KUKA KRL program: EPS_2_25990_SANMH03_A_20251014010956.src

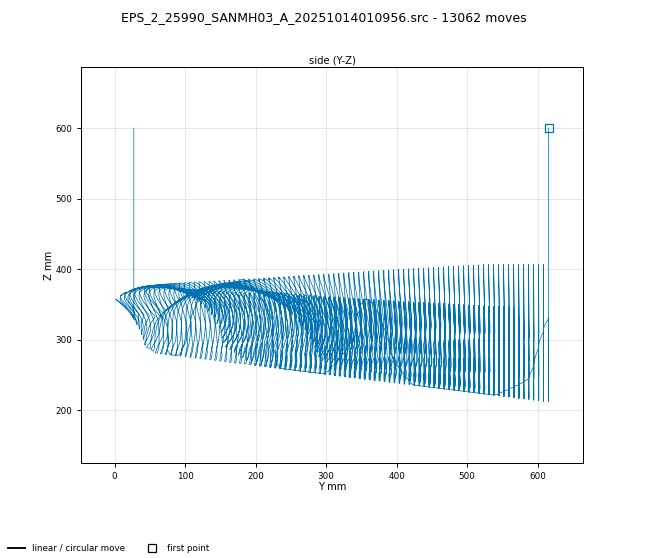
[picture p0: tool path of EPS_2_25990_SANMH03_A_20251014010956.src, 13062 of 13064 moves have a stored position in this frame; points joined in program order, loops and branches not executed]
&ACCESS RVP
&REL 4
&COMMENT QRS 19112012
&PARAM EDITMASK = *
DEF PART()
EXT BAS (BAS_COMMAND :IN,REAL :IN )
INT I
BAS (#INITMOV,0 )

;KUKA QRS Post kuka4.cps  Date:22-06-2017 !

File_ID=2884

QRS_PRE_INIT()

;Init var - Until changes are made in qrs_pre_init
Outlet_Square_prg=0
Inlet_1_Square_prg=0
Inlet_2_Square_prg=0
Inlet_3_Square_prg=0
Inlet_4_Square_prg=0
Inlet_5_Square_prg=0

Outlet_1={X 0.000, Y 531.880, Z 306.500, B 0.000, E1 0.000 }
Inlet_1={X 0.000, Y 536.220, Z 246.500, B 0.000, E1 91.000 }
Inlet_2={X 0.000, Y 540.650, Z 272.000, B 0.000, E1 217.000 }
Outlet_1_type=201
Inlet_1_type=201
Inlet_2_type=150
;QRS#1=Sidecore dimensions
;QRS#2=200-8" PVC SDR 35
;QRS#3=200-8" PVC SDR 35
;QRS#4=150-6" PVC SDR 28
;QRS#5=
;QRS#6=
;QRS#7=
;QRS#8=
;QRS#9=12-08 PSX
;QRS#10=12-08 PSX
;QRS#11=10-06 PSX
;QRS#12=
;QRS#13=
;QRS#14=
;QRS#15=
;QRS#16=1220x127x686 2,25'
;QRS#17=EPS Height
;QRS#18=407
;QRS#19=*
;QRS#20= UPDATED VERSION 22-06-2017
;QRS#21=*
Outlet_Square=0100
Inlet_1_Square=0100
Inlet_2_Square=070
Inlet_3_Square=0
Inlet_4_Square=0
Inlet_5_Square=0
Mill_Square=1
Outlet_Square_Prg=204
Inlet_1_Square_prg=204
Inlet_2_Square_prg=203

QRS_INIT()

$ADVANCE=5

; T1
PTP {E1 173.516,E2 173.516}
PTP {X 0,Y 615.499,A -85,B 0,C 180,E1 173.516,E2 173.516,E3 0,E4 0,E5 0,E6 0}
QRS_SPEED_INIT()
LIN {X 0,Y 615.499,Z 600,A -85,B 0,C 180,E1 173.516,E2 173.516,E3 0,E4 0,E5 0,E6 0} C_VEL
LIN {X 0,Y 615.499,Z 343.49,A -85,B 0,C 180,E1 173.516,E2 173.516} C_VEL
LIN {X 0,Y 615.499,Z 333.343,A -85,B 0,C 180,E1 173.516,E2 173.516} C_VEL
LIN {X 0,Y 615.495,Z 331.594,A -85,B 0,C 180,E1 173.42,E2 173.42} C_VEL
LIN {X 0,Y 615.496,Z 325.468,A -85,B 0,C 180,E1 172.454,E2 172.454} C_VEL
LIN {X 0,Y 615.497,Z 317.616,A -85,B 0,C 180,E1 171.463,E2 171.463} C_VEL
LIN {X 0,Y 615.498,Z 307.826,A -85,B 0,C 180,E1 170.47,E2 170.47} C_VEL
LIN {X 0,Y 615.498,Z 297.546,A -85,B 0,C 180,E1 169.639,E2 169.639} C_VEL
LIN {X 0,Y 615.47,Z 285.87,A -85,B 0,C 180,E1 168.885,E2 168.885} C_VEL
LIN {X 0,Y 615.494,Z 274.386,A -85,B 0,C 180,E1 168.306,E2 168.306} C_VEL
LIN {X 0,Y 615.485,Z 262.385,A -85,B 0,C 180,E1 167.846,E2 167.846} C_VEL
LIN {X 0,Y 615.487,Z 250.236,A -85,B 0,C 180,E1 167.512,E2 167.512} C_VEL
LIN {X 0,Y 615.486,Z 243.189,A -85,B 0,C 180,E1 167.365,E2 167.365} C_VEL
LIN {X 0,Y 615.467,Z 239.503,A -85,B 0,C 180,E1 164.773,E2 164.773} C_VEL
LIN {X 0,Y 615.492,Z 235.664,A -85,B 0,C 180,E1 162.043,E2 162.043} C_VEL
LIN {X 0,Y 615.451,Z 231.833,A -85,B 0,C 180,E1 159.268,E2 159.268} C_VEL
LIN {X 0,Y 615.489,Z 227.979,A -85,B 0,C 180,E1 156.444,E2 156.444} C_VEL
LIN {X 0,Y 615.499,Z 225.095,A -85,B 0,C 180,E1 154.285,E2 154.285} C_VEL
LIN {X 0,Y 615.431,Z 221.535,A -85,B 0,C 180,E1 151.56,E2 151.56} C_VEL
LIN {X 0,Y 615.482,Z 218.202,A -85,B 0,C 180,E1 148.916,E2 148.916} C_VEL
LIN {X 0,Y 615.46,Z 214.61,A -85,B 0,C 180,E1 145.976,E2 145.976} C_VEL
LIN {X 0,Y 615.49,Z 211.697,A -85,B 0,C 180,E1 143.575,E2 143.575} C_VEL
LIN {X 0,Y 615.494,Z 211.683,A -85,B 0,C 180,E1 140.938,E2 140.938} C_VEL
LIN {X 0,Y 615.476,Z 211.697,A -85,B 0,C 180,E1 137.922,E2 137.922} C_VEL
LIN {X 0,Y 615.492,Z 211.687,A -85,B 0,C 180,E1 135.069,E2 135.069} C_VEL
LIN {X 0,Y 615.464,Z 211.698,A -85,B 0,C 180,E1 132.355,E2 132.355} C_VEL
LIN {X 0,Y 615.436,Z 211.697,A -85,B 0,C 180,E1 129.755,E2 129.755} C_VEL
LIN {X 0,Y 615.487,Z 211.699,A -85,B 0,C 180,E1 127.243,E2 127.243} C_VEL
LIN {X 0,Y 615.44,Z 211.698,A -85,B 0,C 180,E1 124.694,E2 124.694} C_VEL
LIN {X 0,Y 615.438,Z 211.697,A -85,B 0,C 180,E1 122.323,E2 122.323} C_VEL
LIN {X 0,Y 615.495,Z 211.7,A -85,B 0,C 180,E1 119.795,E2 119.795} C_VEL
LIN {X 0,Y 615.469,Z 211.689,A -85,B 0,C 180,E1 117.041,E2 117.041} C_VEL
LIN {X 0,Y 615.487,Z 211.702,A -85,B 0,C 180,E1 114.272,E2 114.272} C_VEL
LIN {X 0,Y 615.493,Z 211.684,A -85,B 0,C 180,E1 111.432,E2 111.432} C_VEL
LIN {X 0,Y 615.485,Z 211.699,A -85,B 0,C 180,E1 108.603,E2 108.603} C_VEL
LIN {X 0,Y 615.477,Z 211.687,A -85,B 0,C 180,E1 105.906,E2 105.906} C_VEL
LIN {X 0,Y 615.495,Z 211.701,A -85,B 0,C 180,E1 103.201,E2 103.201} C_VEL
LIN {X 0,Y 615.441,Z 211.696,A -85,B 0,C 180,E1 100.528,E2 100.528} C_VEL
LIN {X 0,Y 615.484,Z 211.697,A -85,B 0,C 180,E1 97.876,E2 97.876} C_VEL
LIN {X 0,Y 615.432,Z 211.7,A -85,B 0,C 180,E1 95.242,E2 95.242} C_VEL
LIN {X 0,Y 615.433,Z 211.698,A -85,B 0,C 180,E1 93.273,E2 93.273} C_VEL
LIN {X 0,Y 615.439,Z 211.696,A -85,B 0,C 180,E1 91.309,E2 91.309} C_VEL
LIN {X 0,Y 615.472,Z 211.699,A -85,B 0,C 180,E1 88.691,E2 88.691} C_VEL
LIN {X 0,Y 615.487,Z 211.688,A -85,B 0,C 180,E1 86.072,E2 86.072} C_VEL
LIN {X 0,Y 615.477,Z 211.777,A -85,B 0,C 180,E1 85.005,E2 85.005} C_VEL
LIN {X 0,Y 615.488,Z 217.2,A -85,B 0,C 180,E1 82.784,E2 82.784} C_VEL
LIN {X 0,Y 615.49,Z 223.43,A -85,B 0,C 180,E1 80.138,E2 80.138} C_VEL
LIN {X 0,Y 615.452,Z 229.574,A -85,B 0,C 180,E1 77.469,E2 77.469} C_VEL
LIN {X 0,Y 615.493,Z 235.878,A -85,B 0,C 180,E1 74.774,E2 74.774} C_VEL
LIN {X 0,Y 615.474,Z 242.411,A -85,B 0,C 180,E1 72.043,E2 72.043} C_VEL
LIN {X 0,Y 615.487,Z 249.137,A -85,B 0,C 180,E1 69.269,E2 69.269} C_VEL
LIN {X 0,Y 615.485,Z 256.099,A -85,B 0,C 180,E1 66.444,E2 66.444} C_VEL
LIN {X 0,Y 615.479,Z 263.285,A -85,B 0,C 180,E1 63.555,E2 63.555} C_VEL
LIN {X 0,Y 615.49,Z 266.918,A -85,B 0,C 180,E1 62.108,E2 62.108} C_VEL
LIN {X 0,Y 615.488,Z 278.231,A -85,B 0,C 180,E1 61.82,E2 61.82} C_VEL
LIN {X 0,Y 615.464,Z 288.228,A -85,B 0,C 180,E1 61.447,E2 61.447} C_VEL
LIN {X 0,Y 615.467,Z 296.234,A -85,B 0,C 180,E1 61.061,E2 61.061} C_VEL
LIN {X 0,Y 615.491,Z 304.039,A -85,B 0,C 180,E1 60.594,E2 60.594} C_VEL
LIN {X 0,Y 615.496,Z 311.816,A -85,B 0,C 180,E1 60.023,E2 60.023} C_VEL
LIN {X 0,Y 615.498,Z 318.16,A -85,B 0,C 180,E1 59.461,E2 59.461} C_VEL
LIN {X 0,Y 615.498,Z 324.688,A -85,B 0,C 180,E1 58.764,E2 58.764} C_VEL
LIN {X 0,Y 615.496,Z 330.585,A -85,B 0,C 180,E1 57.992,E2 57.992} C_VEL
LIN {X 0,Y 615.493,Z 335.716,A -85,B 0,C 180,E1 57.154,E2 57.154} C_VEL
LIN {X 0,Y 615.494,Z 339.016,A -85,B 0,C 180,E1 56.466,E2 56.466} C_VEL
LIN {X 0,Y 615.494,Z 343.165,A -85,B 0,C 180,E1 55.299,E2 55.299} C_VEL
LIN {X 0,Y 615.492,Z 345.468,A -85,B 0,C 180,E1 54.166,E2 54.166} C_VEL
LIN {X 0,Y 615.495,Z 346.361,A -85,B 0,C 180,E1 53.063,E2 53.063} C_VEL
LIN {X 0,Y 615.491,Z 345.737,A -85,B 0,C 180,E1 51.932,E2 51.932} C_VEL
LIN {X 0,Y 615.499,Z 343.952,A -85,B 0,C 180,E1 50.937,E2 50.937} C_VEL
LIN {X 0,Y 615.498,Z 340.875,A -85,B 0,C 180,E1 49.91,E2 49.91} C_VEL
LIN {X 0,Y 615.493,Z 336.533,A -85,B 0,C 180,E1 48.905,E2 48.905} C_VEL
LIN {X 0,Y 615.497,Z 330.597,A -85,B 0,C 180,E1 47.919,E2 47.919} C_VEL
LIN {X 0,Y 615.497,Z 324.524,A -85,B 0,C 180,E1 47.127,E2 47.127} C_VEL
LIN {X 0,Y 615.495,Z 319.388,A -85,B 0,C 180,E1 46.568,E2 46.568} C_VEL
LIN {X 0,Y 615.496,Z 313.223,A -85,B 0,C 180,E1 46.002,E2 46.002} C_VEL
LIN {X 0,Y 615.484,Z 306.158,A -85,B 0,C 180,E1 45.46,E2 45.46} C_VEL
LIN {X 0,Y 615.495,Z 298.933,A -85,B 0,C 180,E1 45.001,E2 45.001} C_VEL
LIN {X 0,Y 615.477,Z 291.057,A -85,B 0,C 180,E1 44.59,E2 44.59} C_VEL
LIN {X 0,Y 615.481,Z 282.81,A -85,B 0,C 180,E1 44.248,E2 44.248} C_VEL
LIN {X 0,Y 615.485,Z 273.161,A -85,B 0,C 180,E1 43.95,E2 43.95} C_VEL
LIN {X 0,Y 615.486,Z 266.876,A -85,B 0,C 180,E1 43.785,E2 43.785} C_VEL
LIN {X 0,Y 615.486,Z 260.138,A -85,B 0,C 180,E1 41.094,E2 41.094} C_VEL
LIN {X 0,Y 615.487,Z 253.669,A -85,B 0,C 180,E1 38.486,E2 38.486} C_VEL
LIN {X 0,Y 615.459,Z 247.171,A -85,B 0,C 180,E1 35.83,E2 35.83} C_VEL
LIN {X 0,Y 615.489,Z 240.885,A -85,B 0,C 180,E1 33.236,E2 33.236} C_VEL
LIN {X 0,Y 615.487,Z 235.37,A -85,B 0,C 180,E1 30.92,E2 30.92} C_VEL
LIN {X 0,Y 615.433,Z 229.578,A -85,B 0,C 180,E1 28.441,E2 28.441} C_VEL
LIN {X 0,Y 615.426,Z 224.987,A -85,B 0,C 180,E1 26.447,E2 26.447} C_VEL
LIN {X 0,Y 615.491,Z 219.28,A -85,B 0,C 180,E1 24.008,E2 24.008} C_VEL
LIN {X 0,Y 615.498,Z 212.782,A -85,B 0,C 180,E1 21.432,E2 21.432} C_VEL
LIN {X 0,Y 615.476,Z 211.7,A -85,B 0,C 180,E1 20.994,E2 20.994} C_VEL
LIN {X 0,Y 615.475,Z 211.7,A -85,B 0,C 180,E1 18.6,E2 18.6} C_VEL
LIN {X 0,Y 615.485,Z 211.696,A -85,B 0,C 180,E1 15.905,E2 15.905} C_VEL
LIN {X 0,Y 615.485,Z 211.699,A -85,B 0,C 180,E1 13.201,E2 13.201} C_VEL
LIN {X 0,Y 615.489,Z 211.701,A -85,B 0,C 180,E1 10.527,E2 10.527} C_VEL
LIN {X 0,Y 615.493,Z 211.696,A -85,B 0,C 180,E1 7.876,E2 7.876} C_VEL
LIN {X 0,Y 615.467,Z 211.7,A -85,B 0,C 180,E1 5.241,E2 5.241} C_VEL
LIN {X 0,Y 615.471,Z 211.7,A -85,B 0,C 180,E1 2.618,E2 2.618} C_VEL
LIN {X 0,Y 615.49,Z 211.7,A -85,B 0,C 180,E1 0,E2 0} C_VEL
LIN {X 0,Y 615.488,Z 211.7,A -85,B 0,C 180,E1 -2.618,E2 -2.618} C_VEL
LIN {X 0,Y 615.478,Z 211.699,A -85,B 0,C 180,E1 -5.241,E2 -5.241} C_VEL
LIN {X 0,Y 615.492,Z 211.695,A -85,B 0,C 180,E1 -7.876,E2 -7.876} C_VEL
LIN {X 0,Y 615.489,Z 211.701,A -85,B 0,C 180,E1 -10.887,E2 -10.887} C_VEL
LIN {X 0,Y 615.49,Z 211.695,A -85,B 0,C 180,E1 -13.932,E2 -13.932} C_VEL
LIN {X 0,Y 615.485,Z 211.7,A -85,B 0,C 180,E1 -16.587,E2 -16.587} C_VEL
LIN {X 0,Y 615.496,Z 211.697,A -85,B 0,C 180,E1 -19.338,E2 -19.338} C_VEL
LIN {X 0,Y 615.472,Z 211.7,A -85,B 0,C 180,E1 -22.342,E2 -22.342} C_VEL
LIN {X 0,Y 615.491,Z 211.7,A -85,B 0,C 180,E1 -24.992,E2 -24.992} C_VEL
LIN {X 0,Y 615.48,Z 211.699,A -85,B 0,C 180,E1 -27.178,E2 -27.178} C_VEL
LIN {X 0,Y 615.498,Z 211.699,A -85,B 0,C 180,E1 -29.796,E2 -29.796} C_VEL
LIN {X 0,Y 615.482,Z 211.699,A -85,B 0,C 180,E1 -32.458,E2 -32.458} C_VEL
LIN {X 0,Y 615.491,Z 211.698,A -85,B 0,C 180,E1 -34.815,E2 -34.815} C_VEL
LIN {X 0,Y 615.493,Z 211.696,A -85,B 0,C 180,E1 -37.242,E2 -37.242} C_VEL
LIN {X 0,Y 615.468,Z 211.7,A -85,B 0,C 180,E1 -40.087,E2 -40.087} C_VEL
LIN {X 0,Y 615.465,Z 211.701,A -85,B 0,C 180,E1 -42.355,E2 -42.355} C_VEL
LIN {X 0,Y 615.497,Z 211.696,A -85,B 0,C 180,E1 -45.068,E2 -45.068} C_VEL
LIN {X 0,Y 615.476,Z 211.701,A -85,B 0,C 180,E1 -47.921,E2 -47.921} C_VEL
LIN {X 0,Y 615.498,Z 211.695,A -85,B 0,C 180,E1 -50.937,E2 -50.937} C_VEL
LIN {X 0,Y 615.486,Z 211.702,A -85,B 0,C 180,E1 -53.575,E2 -53.575} C_VEL
LIN {X 0,Y 615.472,Z 211.749,A -85,B 0,C 180,E1 -54.483,E2 -54.483} C_VEL
LIN {X 0,Y 615.478,Z 220.573,A -85,B 0,C 180,E1 -57.153,E2 -57.153} C_VEL
LIN {X 0,Y 615.453,Z 229.832,A -85,B 0,C 180,E1 -59.838,E2 -59.838} C_VEL
LIN {X 0,Y 615.492,Z 239.075,A -85,B 0,C 180,E1 -62.455,E2 -62.455} C_VEL
LIN {X 0,Y 615.456,Z 248.32,A -85,B 0,C 180,E1 -65.007,E2 -65.007} C_VEL
LIN {X 0,Y 615.473,Z 258.107,A -85,B 0,C 180,E1 -67.658,E2 -67.658} C_VEL
LIN {X 0,Y 615.487,Z 268.102,A -85,B 0,C 180,E1 -70.315,E2 -70.315} C_VEL
LIN {X 0,Y 615.486,Z 278.641,A -85,B 0,C 180,E1 -73.072,E2 -73.072} C_VEL
LIN {X 0,Y 615.464,Z 289.077,A -85,B 0,C 180,E1 -75.761,E2 -75.761} C_VEL
LIN {X 0,Y 615.498,Z 299.209,A -85,B 0,C 180,E1 -78.348,E2 -78.348} C_VEL
LIN {X 0,Y 615.497,Z 313.822,A -85,B 0,C 180,E1 -78.64,E2 -78.64} C_VEL
LIN {X 0,Y 615.453,Z 326.972,A -85,B 0,C 180,E1 -79.051,E2 -79.051} C_VEL
LIN {X 0,Y 615.442,Z 338.774,A -85,B 0,C 180,E1 -79.556,E2 -79.556} C_VEL
LIN {X 0,Y 615.489,Z 349.388,A -85,B 0,C 180,E1 -80.138,E2 -80.138} C_VEL
LIN {X 0,Y 615.498,Z 360.232,A -85,B 0,C 180,E1 -80.884,E2 -80.884} C_VEL
LIN {X 0,Y 615.497,Z 370.812,A -85,B 0,C 180,E1 -81.794,E2 -81.794} C_VEL
LIN {X 0,Y 615.498,Z 378.607,A -85,B 0,C 180,E1 -82.62,E2 -82.62} C_VEL
LIN {X 0,Y 615.496,Z 386.203,A -85,B 0,C 180,E1 -83.608,E2 -83.608} C_VEL
LIN {X 0,Y 615.498,Z 393.205,A -85,B 0,C 180,E1 -84.759,E2 -84.759} C_VEL
LIN {X 0,Y 615.494,Z 397.852,A -85,B 0,C 180,E1 -85.744,E2 -85.744} C_VEL
LIN {X 0,Y 615.494,Z 401.399,A -85,B 0,C 180,E1 -86.727,E2 -86.727} C_VEL
LIN {X 0,Y 615.497,Z 403.233,A -85,B 0,C 180,E1 -87.382,E2 -87.382} C_VEL
LIN {X 0,Y 615.5,Z 404.608,A -85,B 0,C 180,E1 -88.037,E2 -88.037} C_VEL
LIN {X 0,Y 615.496,Z 406.174,A -85,B 0,C 180,E1 -89.346,E2 -89.346} C_VEL
LIN {X 0,Y 615.494,Z 406.389,A -85,B 0,C 180,E1 -90,E2 -90} C_VEL
LIN {X 0,Y 615.495,Z 405.58,A -85,B 0,C 180,E1 -91.309,E2 -91.309} C_VEL
LIN {X 0,Y 615.5,Z 404.607,A -85,B 0,C 180,E1 -91.963,E2 -91.963} C_VEL
LIN {X 0,Y 615.497,Z 403.233,A -85,B 0,C 180,E1 -92.618,E2 -92.618} C_VEL
LIN {X 0,Y 615.496,Z 400.349,A -85,B 0,C 180,E1 -93.601,E2 -93.601} C_VEL
LIN {X 0,Y 615.498,Z 396.441,A -85,B 0,C 180,E1 -94.585,E2 -94.585} C_VEL
LIN {X 0,Y 615.499,Z 391.404,A -85,B 0,C 180,E1 -95.57,E2 -95.57} C_VEL
LIN {X 0,Y 615.497,Z 384.869,A -85,B 0,C 180,E1 -96.583,E2 -96.583} C_VEL
LIN {X 0,Y 615.497,Z 377.132,A -85,B 0,C 180,E1 -97.546,E2 -97.546} C_VEL
LIN {X 0,Y 615.498,Z 369.043,A -85,B 0,C 180,E1 -98.371,E2 -98.371} C_VEL
LIN {X 0,Y 615.499,Z 359.165,A -85,B 0,C 180,E1 -99.199,E2 -99.199} C_VEL
LIN {X 0,Y 615.479,Z 347.98,A -85,B 0,C 180,E1 -99.946,E2 -99.946} C_VEL
LIN {X 0,Y 615.441,Z 337.026,A -85,B 0,C 180,E1 -100.528,E2 -100.528} C_VEL
LIN {X 0,Y 615.459,Z 324.774,A -85,B 0,C 180,E1 -101.031,E2 -101.031} C_VEL
LIN {X 0,Y 615.498,Z 312.055,A -85,B 0,C 180,E1 -101.402,E2 -101.402} C_VEL
LIN {X 0,Y 615.498,Z 299.208,A -85,B 0,C 180,E1 -101.652,E2 -101.652} C_VEL
LIN {X 0,Y 615.464,Z 289.077,A -85,B 0,C 180,E1 -104.239,E2 -104.239} C_VEL
LIN {X 0,Y 615.486,Z 278.64,A -85,B 0,C 180,E1 -106.929,E2 -106.929} C_VEL
LIN {X 0,Y 615.487,Z 268.101,A -85,B 0,C 180,E1 -109.685,E2 -109.685} C_VEL
LIN {X 0,Y 615.476,Z 258.104,A -85,B 0,C 180,E1 -112.343,E2 -112.343} C_VEL
LIN {X 0,Y 615.456,Z 248.32,A -85,B 0,C 180,E1 -114.993,E2 -114.993} C_VEL
LIN {X 0,Y 615.448,Z 237.758,A -85,B 0,C 180,E1 -117.917,E2 -117.917} C_VEL
LIN {X 0,Y 615.464,Z 228.484,A -85,B 0,C 180,E1 -120.541,E2 -120.541} C_VEL
LIN {X 0,Y 615.486,Z 220.546,A -85,B 0,C 180,E1 -122.846,E2 -122.846} C_VEL
LIN {X 0,Y 615.492,Z 213.086,A -85,B 0,C 180,E1 -125.215,E2 -125.215} C_VEL
LIN {X 0,Y 615.47,Z 211.7,A -85,B 0,C 180,E1 -125.724,E2 -125.724} C_VEL
LIN {X 0,Y 615.479,Z 211.701,A -85,B 0,C 180,E1 -128.07,E2 -128.07} C_VEL
LIN {X 0,Y 615.488,Z 211.694,A -85,B 0,C 180,E1 -131.094,E2 -131.094} C_VEL
LIN {X 0,Y 615.482,Z 211.7,A -85,B 0,C 180,E1 -133.997,E2 -133.997} C_VEL
LIN {X 0,Y 615.492,Z 211.697,A -85,B 0,C 180,E1 -136.953,E2 -136.953} C_VEL
LIN {X 0,Y 615.48,Z 211.701,A -85,B 0,C 180,E1 -139.393,E2 -139.393} C_VEL
LIN {X 0,Y 615.483,Z 211.699,A -85,B 0,C 180,E1 -141.989,E2 -141.989} C_VEL
LIN {X 0,Y 615.496,Z 211.699,A -85,B 0,C 180,E1 -144.385,E2 -144.385} C_VEL
LIN {X 0,Y 615.487,Z 211.698,A -85,B 0,C 180,E1 -145.3,E2 -145.3} C_VEL
LIN {X 0,Y 615.466,Z 214.459,A -85,B 0,C 180,E1 -147.673,E2 -147.673} C_VEL
LIN {X 0,Y 615.453,Z 217.446,A -85,B 0,C 180,E1 -150.212,E2 -150.212} C_VEL
LIN {X 0,Y 615.448,Z 220.642,A -85,B 0,C 180,E1 -152.963,E2 -152.963} C_VEL
LIN {X 0,Y 615.445,Z 223.297,A -85,B 0,C 180,E1 -155.006,E2 -155.006} C_VEL
LIN {X 0,Y 615.436,Z 226.139,A -85,B 0,C 180,E1 -157.153,E2 -157.153} C_VEL
LIN {X 0,Y 615.435,Z 229.243,A -85,B 0,C 180,E1 -159.457,E2 -159.457} C_VEL
LIN {X 0,Y 615.494,Z 232.768,A -85,B 0,C 180,E1 -162.043,E2 -162.043} C_VEL
LIN {X 0,Y 615.458,Z 236.563,A -85,B 0,C 180,E1 -164.773,E2 -164.773} C_VEL
LIN {X 0,Y 615.474,Z 240.371,A -85,B 0,C 180,E1 -167.47,E2 -167.47} C_VEL
LIN {X 0,Y 615.484,Z 243.185,A -85,B 0,C 180,E1 -169.451,E2 -169.451} C_VEL
LIN {X 0,Y 615.487,Z 258.21,A -85,B 0,C 180,E1 -169.806,E2 -169.806} C_VEL
LIN {X 0,Y 615.491,Z 270.248,A -85,B 0,C 180,E1 -170.221,E2 -170.221} C_VEL
LIN {X 0,Y 615.463,Z 282.68,A -85,B 0,C 180,E1 -170.801,E2 -170.801} C_VEL
LIN {X 0,Y 615.49,Z 293.753,A -85,B 0,C 180,E1 -171.463,E2 -171.463} C_VEL
LIN {X 0,Y 615.498,Z 302.72,A -85,B 0,C 180,E1 -172.125,E2 -172.125} C_VEL
LIN {X 0,Y 615.499,Z 311.875,A -85,B 0,C 180,E1 -172.943,E2 -172.943} C_VEL
LIN {X 0,Y 615.497,Z 320.848,A -85,B 0,C 180,E1 -173.937,E2 -173.937} C_VEL
LIN {X 0,Y 615.497,Z 328.03,A -85,B 0,C 180,E1 -174.923,E2 -174.923} C_VEL
LIN {X 0,Y 615.493,Z 332.875,A -85,B 0,C 180,E1 -175.744,E2 -175.744} C_VEL
LIN {X 0,Y 615.496,Z 337.586,A -85,B 0,C 180,E1 -176.727,E2 -176.727} C_VEL
LIN {X 0,Y 615.498,Z 341.198,A -85,B 0,C 180,E1 -177.71,E2 -177.71} C_VEL
LIN {X 0,Y 615.496,Z 343.818,A -85,B 0,C 180,E1 -178.691,E2 -178.691} C_VEL
LIN {X 0,Y 615.497,Z 345.889,A -85,B 0,C 180,E1 -180,E2 -180} C_VEL
LIN {X 0,Y 615.496,Z 346.331,A -85,B 0,C 180,E1 -181.309,E2 -181.309} C_VEL
LIN {X 0,Y 615.495,Z 345.257,A -85,B 0,C 180,E1 -182.618,E2 -182.618} C_VEL
LIN {X 0,Y 615.496,Z 344.09,A -85,B 0,C 180,E1 -183.273,E2 -183.273} C_VEL
LIN {X 0,Y 615.495,Z 342.523,A -85,B 0,C 180,E1 -183.929,E2 -183.929} C_VEL
LIN {X 0,Y 615.494,Z 339.368,A -85,B 0,C 180,E1 -184.913,E2 -184.913} C_VEL
LIN {X 0,Y 615.499,Z 335.16,A -85,B 0,C 180,E1 -185.899,E2 -185.899} C_VEL
LIN {X 0,Y 615.495,Z 331.594,A -85,B 0,C 180,E1 -186.58,E2 -186.58} C_VEL
LIN {X 0,Y 614.823,Z 328.889,A -85,B 0,C 180,E1 -187.058,E2 -187.058} C_VEL
LIN {X 0,Y 611.98,Z 324.085,A -85,B 0,C 180,E1 -187.824,E2 -187.824} C_VEL
LIN {X 0,Y 609.133,Z 318.554,A -85,B 0,C 180,E1 -188.557,E2 -188.557} C_VEL
LIN {X 0,Y 608.473,Z 314.714,A -85,B 0,C 180,E1 -188.981,E2 -188.981} C_VEL
LIN {X 0,Y 608.488,Z 306.05,A -85,B 0,C 180,E1 -189.809,E2 -189.809} C_VEL
LIN {X 0,Y 608.493,Z 295.27,A -85,B 0,C 180,E1 -190.649,E2 -190.649} C_VEL
LIN {X 0,Y 608.474,Z 284.411,A -85,B 0,C 180,E1 -191.324,E2 -191.324} C_VEL
LIN {X 0,Y 608.51,Z 272.262,A -85,B 0,C 180,E1 -191.914,E2 -191.914} C_VEL
LIN {X 0,Y 608.528,Z 259.521,A -85,B 0,C 180,E1 -192.379,E2 -192.379} C_VEL
LIN {X 0,Y 608.545,Z 246.819,A -85,B 0,C 180,E1 -192.697,E2 -192.697} C_VEL
LIN {X 0,Y 608.41,Z 243.681,A -85,B 0,C 180,E1 -192.763,E2 -192.763} C_VEL
LIN {X 0,Y 608.41,Z 240.906,A -85,B 0,C 180,E1 -194.722,E2 -194.722} C_VEL
LIN {X 0,Y 608.401,Z 237.042,A -85,B 0,C 180,E1 -197.478,E2 -197.478} C_VEL
LIN {X 0,Y 608.417,Z 233.175,A -85,B 0,C 180,E1 -200.276,E2 -200.276} C_VEL
LIN {X 0,Y 608.397,Z 229.303,A -85,B 0,C 180,E1 -203.126,E2 -203.126} C_VEL
LIN {X 0,Y 608.405,Z 225.427,A -85,B 0,C 180,E1 -206.038,E2 -206.038} C_VEL
LIN {X 0,Y 608.374,Z 222.091,A -85,B 0,C 180,E1 -208.602,E2 -208.602} C_VEL
LIN {X 0,Y 608.416,Z 218.808,A -85,B 0,C 180,E1 -211.262,E2 -211.262} C_VEL
LIN {X 0,Y 608.429,Z 215.796,A -85,B 0,C 180,E1 -213.728,E2 -213.728} C_VEL
LIN {X 0,Y 608.449,Z 212.93,A -85,B 0,C 180,E1 -216.092,E2 -216.092} C_VEL
LIN {X 0,Y 608.472,Z 212.694,A -85,B 0,C 180,E1 -218.24,E2 -218.24} C_VEL
LIN {X 0,Y 608.464,Z 212.69,A -85,B 0,C 180,E1 -221.342,E2 -221.342} C_VEL
LIN {X 0,Y 608.458,Z 212.694,A -85,B 0,C 180,E1 -223.871,E2 -223.871} C_VEL
LIN {X 0,Y 608.465,Z 212.688,A -85,B 0,C 180,E1 -226.692,E2 -226.692} C_VEL
LIN {X 0,Y 608.421,Z 212.695,A -85,B 0,C 180,E1 -229.694,E2 -229.694} C_VEL
LIN {X 0,Y 608.431,Z 212.692,A -85,B 0,C 180,E1 -232.251,E2 -232.251} C_VEL
LIN {X 0,Y 608.416,Z 212.696,A -85,B 0,C 180,E1 -235.1,E2 -235.1} C_VEL
LIN {X 0,Y 608.422,Z 212.693,A -85,B 0,C 180,E1 -237.484,E2 -237.484} C_VEL
LIN {X 0,Y 608.479,Z 212.695,A -85,B 0,C 180,E1 -240.221,E2 -240.221} C_VEL
LIN {X 0,Y 608.43,Z 212.692,A -85,B 0,C 180,E1 -243.225,E2 -243.225} C_VEL
LIN {X 0,Y 608.482,Z 212.693,A -85,B 0,C 180,E1 -245.848,E2 -245.848} C_VEL
LIN {X 0,Y 608.472,Z 212.687,A -85,B 0,C 180,E1 -248.308,E2 -248.308} C_VEL
LIN {X 0,Y 608.473,Z 212.696,A -85,B 0,C 180,E1 -251.285,E2 -251.285} C_VEL
LIN {X 0,Y 608.449,Z 212.689,A -85,B 0,C 180,E1 -253.906,E2 -253.906} C_VEL
LIN {X 0,Y 608.469,Z 212.693,A -85,B 0,C 180,E1 -256.644,E2 -256.644} C_VEL
LIN {X 0,Y 608.424,Z 212.693,A -85,B 0,C 180,E1 -259.349,E2 -259.349} C_VEL
LIN {X 0,Y 608.47,Z 212.691,A -85,B 0,C 180,E1 -262.033,E2 -262.033} C_VEL
LIN {X 0,Y 608.42,Z 212.695,A -85,B 0,C 180,E1 -264.698,E2 -264.698} C_VEL
LIN {X 0,Y 608.438,Z 212.693,A -85,B 0,C 180,E1 -267.352,E2 -267.352} C_VEL
LIN {X 0,Y 608.478,Z 212.69,A -85,B 0,C 180,E1 -270,E2 -270} C_VEL
LIN {X 0,Y 608.449,Z 212.69,A -85,B 0,C 180,E1 -272.648,E2 -272.648} C_VEL
LIN {X 0,Y 608.462,Z 212.811,A -85,B 0,C 180,E1 -275.053,E2 -275.053} C_VEL
LIN {X 0,Y 608.452,Z 219.911,A -85,B 0,C 180,E1 -277.967,E2 -277.967} C_VEL
LIN {X 0,Y 608.405,Z 226.17,A -85,B 0,C 180,E1 -280.651,E2 -280.651} C_VEL
LIN {X 0,Y 608.45,Z 232.381,A -85,B 0,C 180,E1 -283.357,E2 -283.357} C_VEL
LIN {X 0,Y 608.432,Z 238.803,A -85,B 0,C 180,E1 -286.095,E2 -286.095} C_VEL
LIN {X 0,Y 608.434,Z 245.433,A -85,B 0,C 180,E1 -288.87,E2 -288.87} C_VEL
LIN {X 0,Y 608.419,Z 252.287,A -85,B 0,C 180,E1 -291.693,E2 -291.693} C_VEL
LIN {X 0,Y 608.42,Z 259.371,A -85,B 0,C 180,E1 -294.573,E2 -294.573} C_VEL
LIN {X 0,Y 608.435,Z 266.702,A -85,B 0,C 180,E1 -297.519,E2 -297.519} C_VEL
LIN {X 0,Y 608.423,Z 267.347,A -85,B 0,C 180,E1 -297.776,E2 -297.776} C_VEL
LIN {X 0,Y 608.489,Z 279.908,A -85,B 0,C 180,E1 -298.124,E2 -298.124} C_VEL
LIN {X 0,Y 608.469,Z 288.829,A -85,B 0,C 180,E1 -298.467,E2 -298.467} C_VEL
LIN {X 0,Y 608.472,Z 297.332,A -85,B 0,C 180,E1 -298.889,E2 -298.889} C_VEL
LIN {X 0,Y 608.48,Z 305.565,A -85,B 0,C 180,E1 -299.398,E2 -299.398} C_VEL
LIN {X 0,Y 608.458,Z 313.099,A -85,B 0,C 180,E1 -299.969,E2 -299.969} C_VEL
LIN {X 0,Y 608.464,Z 321.362,A -85,B 0,C 180,E1 -300.738,E2 -300.738} C_VEL
LIN {X 0,Y 608.44,Z 327.97,A -85,B 0,C 180,E1 -301.512,E2 -301.512} C_VEL
LIN {X 0,Y 608.453,Z 333.398,A -85,B 0,C 180,E1 -302.305,E2 -302.305} C_VEL
LIN {X 0,Y 608.431,Z 336.709,A -85,B 0,C 180,E1 -302.881,E2 -302.881} C_VEL
LIN {X 0,Y 608.43,Z 340.598,A -85,B 0,C 180,E1 -303.728,E2 -303.728} C_VEL
LIN {X 0,Y 608.424,Z 343.19,A -85,B 0,C 180,E1 -304.472,E2 -304.472} C_VEL
LIN {X 0,Y 608.418,Z 345.211,A -85,B 0,C 180,E1 -305.279,E2 -305.279} C_VEL
LIN {X 0,Y 608.422,Z 346.463,A -85,B 0,C 180,E1 -306.094,E2 -306.094} C_VEL
LIN {X 0,Y 608.437,Z 346.973,A -85,B 0,C 180,E1 -307.154,E2 -307.154} C_VEL
LIN {X 0,Y 608.419,Z 346.125,A -85,B 0,C 180,E1 -308.234,E2 -308.234} C_VEL
LIN {X 0,Y 608.425,Z 344.049,A -85,B 0,C 180,E1 -309.292,E2 -309.292} C_VEL
LIN {X 0,Y 608.436,Z 340.731,A -85,B 0,C 180,E1 -310.327,E2 -310.327} C_VEL
LIN {X 0,Y 608.432,Z 335.974,A -85,B 0,C 180,E1 -311.338,E2 -311.338} C_VEL
LIN {X 0,Y 608.436,Z 331.618,A -85,B 0,C 180,E1 -312.064,E2 -312.064} C_VEL
LIN {X 0,Y 608.468,Z 326.279,A -85,B 0,C 180,E1 -312.788,E2 -312.788} C_VEL
LIN {X 0,Y 608.453,Z 319.239,A -85,B 0,C 180,E1 -313.561,E2 -313.561} C_VEL
LIN {X 0,Y 608.48,Z 312.051,A -85,B 0,C 180,E1 -314.207,E2 -314.207} C_VEL
LIN {X 0,Y 608.461,Z 304.051,A -85,B 0,C 180,E1 -314.796,E2 -314.796} C_VEL
LIN {X 0,Y 608.46,Z 293.173,A -85,B 0,C 180,E1 -315.426,E2 -315.426} C_VEL
LIN {X 0,Y 608.501,Z 282.678,A -85,B 0,C 180,E1 -315.869,E2 -315.869} C_VEL
LIN {X 0,Y 608.501,Z 273.542,A -85,B 0,C 180,E1 -316.154,E2 -316.154} C_VEL
LIN {X 0,Y 608.442,Z 267.33,A -85,B 0,C 180,E1 -316.32,E2 -316.32} C_VEL
LIN {X 0,Y 608.425,Z 260.011,A -85,B 0,C 180,E1 -319.259,E2 -319.259} C_VEL
LIN {X 0,Y 608.416,Z 253.831,A -85,B 0,C 180,E1 -321.766,E2 -321.766} C_VEL
LIN {X 0,Y 608.409,Z 248.481,A -85,B 0,C 180,E1 -323.96,E2 -323.96} C_VEL
LIN {X 0,Y 608.413,Z 242.779,A -85,B 0,C 180,E1 -326.326,E2 -326.326} C_VEL
LIN {X 0,Y 608.449,Z 237.061,A -85,B 0,C 180,E1 -328.733,E2 -328.733} C_VEL
LIN {X 0,Y 608.398,Z 230.857,A -85,B 0,C 180,E1 -331.394,E2 -331.394} C_VEL
LIN {X 0,Y 608.404,Z 226.661,A -85,B 0,C 180,E1 -333.223,E2 -333.223} C_VEL
LIN {X 0,Y 608.46,Z 220.468,A -85,B 0,C 180,E1 -335.852,E2 -335.852} C_VEL
LIN {X 0,Y 608.458,Z 213.38,A -85,B 0,C 180,E1 -338.664,E2 -338.664} C_VEL
LIN {X 0,Y 608.458,Z 212.695,A -85,B 0,C 180,E1 -339.018,E2 -339.018} C_VEL
LIN {X 0,Y 608.44,Z 212.696,A -85,B 0,C 180,E1 -341.828,E2 -341.828} C_VEL
LIN {X 0,Y 608.471,Z 212.695,A -85,B 0,C 180,E1 -344.594,E2 -344.594} C_VEL
LIN {X 0,Y 608.464,Z 212.694,A -85,B 0,C 180,E1 -347.323,E2 -347.323} C_VEL
LIN {X 0,Y 608.464,Z 212.693,A -85,B 0,C 180,E1 -350.023,E2 -350.023} C_VEL
LIN {X 0,Y 608.468,Z 212.694,A -85,B 0,C 180,E1 -352.701,E2 -352.701} C_VEL
LIN {X 0,Y 608.461,Z 212.697,A -85,B 0,C 180,E1 -355.362,E2 -355.362} C_VEL
LIN {X 0,Y 608.469,Z 212.694,A -85,B 0,C 180,E1 -358.014,E2 -358.014} C_VEL
LIN {X 0,Y 608.464,Z 212.693,A -85,B 0,C 180,E1 -360.662,E2 -360.662} C_VEL
LIN {X 0,Y 608.466,Z 212.693,A -85,B 0,C 180,E1 -363.311,E2 -363.311} C_VEL
LIN {X 0,Y 608.469,Z 212.695,A -85,B 0,C 180,E1 -365.967,E2 -365.967} C_VEL
LIN {X 0,Y 608.453,Z 212.696,A -85,B 0,C 180,E1 -368.636,E2 -368.636} C_VEL
LIN {X 0,Y 608.46,Z 212.693,A -85,B 0,C 180,E1 -371.324,E2 -371.324} C_VEL
LIN {X 0,Y 608.473,Z 212.692,A -85,B 0,C 180,E1 -374.037,E2 -374.037} C_VEL
LIN {X 0,Y 608.459,Z 212.697,A -85,B 0,C 180,E1 -376.784,E2 -376.784} C_VEL
LIN {X 0,Y 608.458,Z 212.694,A -85,B 0,C 180,E1 -379.57,E2 -379.57} C_VEL
LIN {X 0,Y 608.462,Z 212.695,A -85,B 0,C 180,E1 -382.476,E2 -382.476} C_VEL
LIN {X 0,Y 608.452,Z 212.696,A -85,B 0,C 180,E1 -385.301,E2 -385.301} C_VEL
LIN {X 0,Y 608.441,Z 212.699,A -85,B 0,C 180,E1 -387.518,E2 -387.518} C_VEL
LIN {X 0,Y 608.453,Z 212.697,A -85,B 0,C 180,E1 -389.969,E2 -389.969} C_VEL
LIN {X 0,Y 608.459,Z 212.694,A -85,B 0,C 180,E1 -392.88,E2 -392.88} C_VEL
LIN {X 0,Y 608.449,Z 212.695,A -85,B 0,C 180,E1 -395.277,E2 -395.277} C_VEL
LIN {X 0,Y 608.473,Z 212.692,A -85,B 0,C 180,E1 -397.746,E2 -397.746} C_VEL
LIN {X 0,Y 608.445,Z 212.697,A -85,B 0,C 180,E1 -400.328,E2 -400.328} C_VEL
LIN {X 0,Y 608.473,Z 212.692,A -85,B 0,C 180,E1 -403.309,E2 -403.309} C_VEL
LIN {X 0,Y 608.458,Z 212.694,A -85,B 0,C 180,E1 -406.129,E2 -406.129} C_VEL
LIN {X 0,Y 608.452,Z 212.698,A -85,B 0,C 180,E1 -408.823,E2 -408.823} C_VEL
LIN {X 0,Y 608.441,Z 212.698,A -85,B 0,C 180,E1 -411.41,E2 -411.41} C_VEL
LIN {X 0,Y 608.444,Z 212.697,A -85,B 0,C 180,E1 -413.955,E2 -413.955} C_VEL
LIN {X 0,Y 608.462,Z 212.745,A -85,B 0,C 180,E1 -414.317,E2 -414.317} C_VEL
LIN {X 0,Y 608.524,Z 220.581,A -85,B 0,C 180,E1 -416.73,E2 -416.73} C_VEL
LIN {X 0,Y 608.499,Z 229.832,A -85,B 0,C 180,E1 -419.457,E2 -419.457} C_VEL
LIN {X 0,Y 608.466,Z 239.127,A -85,B 0,C 180,E1 -422.109,E2 -422.109} C_VEL
LIN {X 0,Y 608.472,Z 248.394,A -85,B 0,C 180,E1 -424.7,E2 -424.7} C_VEL
LIN {X 0,Y 608.462,Z 258.986,A -85,B 0,C 180,E1 -427.594,E2 -427.594} C_VEL
LIN {X 0,Y 608.459,Z 269.577,A -85,B 0,C 180,E1 -430.43,E2 -430.43} C_VEL
LIN {X 0,Y 608.452,Z 280.168,A -85,B 0,C 180,E1 -433.216,E2 -433.216} C_VEL
LIN {X 0,Y 608.44,Z 290.889,A -85,B 0,C 180,E1 -435.995,E2 -435.995} C_VEL
LIN {X 0,Y 608.438,Z 299.572,A -85,B 0,C 180,E1 -438.222,E2 -438.222} C_VEL
LIN {X 0,Y 608.549,Z 313.096,A -85,B 0,C 180,E1 -438.488,E2 -438.488} C_VEL
LIN {X 0,Y 608.487,Z 325.517,A -85,B 0,C 180,E1 -438.865,E2 -438.865} C_VEL
LIN {X 0,Y 608.466,Z 337.173,A -85,B 0,C 180,E1 -439.35,E2 -439.35} C_VEL
LIN {X 0,Y 608.479,Z 349.579,A -85,B 0,C 180,E1 -440.023,E2 -440.023} C_VEL
LIN {X 0,Y 608.483,Z 360.475,A -85,B 0,C 180,E1 -440.778,E2 -440.778} C_VEL
LIN {X 0,Y 608.475,Z 371.112,A -85,B 0,C 180,E1 -441.699,E2 -441.699} C_VEL
LIN {X 0,Y 608.471,Z 378.961,A -85,B 0,C 180,E1 -442.534,E2 -442.534} C_VEL
LIN {X 0,Y 608.461,Z 386.287,A -85,B 0,C 180,E1 -443.485,E2 -443.485} C_VEL
LIN {X 0,Y 608.451,Z 391.866,A -85,B 0,C 180,E1 -444.366,E2 -444.366} C_VEL
LIN {X 0,Y 608.432,Z 396.95,A -85,B 0,C 180,E1 -445.362,E2 -445.362} C_VEL
LIN {X 0,Y 608.449,Z 400.896,A -85,B 0,C 180,E1 -446.358,E2 -446.358} C_VEL
LIN {X 0,Y 608.425,Z 403.809,A -85,B 0,C 180,E1 -447.352,E2 -447.352} C_VEL
LIN {X 0,Y 608.445,Z 405.201,A -85,B 0,C 180,E1 -448.014,E2 -448.014} C_VEL
LIN {X 0,Y 608.438,Z 406.784,A -85,B 0,C 180,E1 -449.338,E2 -449.338} C_VEL
LIN {X 0,Y 608.434,Z 407,A -85,B 0,C 180,E1 -450,E2 -450} C_VEL
LIN {X 0,Y 608.448,Z 406.184,A -85,B 0,C 180,E1 -451.324,E2 -451.324} C_VEL
LIN {X 0,Y 608.445,Z 405.201,A -85,B 0,C 180,E1 -451.986,E2 -451.986} C_VEL
LIN {X 0,Y 608.425,Z 403.809,A -85,B 0,C 180,E1 -452.648,E2 -452.648} C_VEL
LIN {X 0,Y 608.449,Z 400.896,A -85,B 0,C 180,E1 -453.643,E2 -453.643} C_VEL
LIN {X 0,Y 608.432,Z 396.949,A -85,B 0,C 180,E1 -454.638,E2 -454.638} C_VEL
LIN {X 0,Y 608.438,Z 390.876,A -85,B 0,C 180,E1 -455.801,E2 -455.801} C_VEL
LIN {X 0,Y 608.462,Z 384.234,A -85,B 0,C 180,E1 -456.799,E2 -456.799} C_VEL
LIN {X 0,Y 608.456,Z 375.988,A -85,B 0,C 180,E1 -457.8,E2 -457.8} C_VEL
LIN {X 0,Y 608.472,Z 367.534,A -85,B 0,C 180,E1 -458.636,E2 -458.636} C_VEL
LIN {X 0,Y 608.481,Z 357.088,A -85,B 0,C 180,E1 -459.474,E2 -459.474} C_VEL
LIN {X 0,Y 608.488,Z 346.753,A -85,B 0,C 180,E1 -460.145,E2 -460.145} C_VEL
LIN {X 0,Y 608.466,Z 335.855,A -85,B 0,C 180,E1 -460.713,E2 -460.713} C_VEL
LIN {X 0,Y 608.493,Z 324.084,A -85,B 0,C 180,E1 -461.186,E2 -461.186} C_VEL
LIN {X 0,Y 608.551,Z 311.258,A -85,B 0,C 180,E1 -461.555,E2 -461.555} C_VEL
LIN {X 0,Y 608.442,Z 299.529,A -85,B 0,C 180,E1 -461.789,E2 -461.789} C_VEL
LIN {X 0,Y 608.433,Z 289.435,A -85,B 0,C 180,E1 -464.38,E2 -464.38} C_VEL
LIN {X 0,Y 608.445,Z 278.843,A -85,B 0,C 180,E1 -467.13,E2 -467.13} C_VEL
LIN {X 0,Y 608.459,Z 269.576,A -85,B 0,C 180,E1 -469.571,E2 -469.571} C_VEL
LIN {X 0,Y 608.463,Z 258.724,A -85,B 0,C 180,E1 -472.476,E2 -472.476} C_VEL
LIN {X 0,Y 608.472,Z 248.394,A -85,B 0,C 180,E1 -475.3,E2 -475.3} C_VEL
LIN {X 0,Y 608.466,Z 239.126,A -85,B 0,C 180,E1 -477.891,E2 -477.891} C_VEL
LIN {X 0,Y 608.465,Z 229.734,A -85,B 0,C 180,E1 -480.545,E2 -480.545} C_VEL
LIN {X 0,Y 608.526,Z 221.822,A -85,B 0,C 180,E1 -482.876,E2 -482.876} C_VEL
LIN {X 0,Y 608.549,Z 214.435,A -85,B 0,C 180,E1 -485.271,E2 -485.271} C_VEL
LIN {X 0,Y 608.434,Z 212.697,A -85,B 0,C 180,E1 -485.919,E2 -485.919} C_VEL
LIN {X 0,Y 608.462,Z 212.694,A -85,B 0,C 180,E1 -488.239,E2 -488.239} C_VEL
LIN {X 0,Y 608.466,Z 212.693,A -85,B 0,C 180,E1 -491.342,E2 -491.342} C_VEL
LIN {X 0,Y 608.464,Z 212.696,A -85,B 0,C 180,E1 -494.264,E2 -494.264} C_VEL
LIN {X 0,Y 608.457,Z 212.695,A -85,B 0,C 180,E1 -497.04,E2 -497.04} C_VEL
LIN {X 0,Y 608.457,Z 212.694,A -85,B 0,C 180,E1 -499.697,E2 -499.697} C_VEL
LIN {X 0,Y 608.47,Z 212.692,A -85,B 0,C 180,E1 -502.254,E2 -502.254} C_VEL
LIN {X 0,Y 608.452,Z 212.695,A -85,B 0,C 180,E1 -505.095,E2 -505.095} C_VEL
LIN {X 0,Y 608.442,Z 212.758,A -85,B 0,C 180,E1 -505.529,E2 -505.529} C_VEL
LIN {X 0,Y 608.412,Z 215.639,A -85,B 0,C 180,E1 -507.902,E2 -507.902} C_VEL
LIN {X 0,Y 608.42,Z 218.34,A -85,B 0,C 180,E1 -510.218,E2 -510.218} C_VEL
LIN {X 0,Y 608.371,Z 221.749,A -85,B 0,C 180,E1 -513.222,E2 -513.222} C_VEL
LIN {X 0,Y 608.382,Z 224.606,A -85,B 0,C 180,E1 -515.426,E2 -515.426} C_VEL
LIN {X 0,Y 608.403,Z 228.42,A -85,B 0,C 180,E1 -518.306,E2 -518.306} C_VEL
LIN {X 0,Y 608.379,Z 232.238,A -85,B 0,C 180,E1 -521.128,E2 -521.128} C_VEL
LIN {X 0,Y 608.442,Z 236.059,A -85,B 0,C 180,E1 -523.906,E2 -523.906} C_VEL
LIN {X 0,Y 608.411,Z 239.885,A -85,B 0,C 180,E1 -526.642,E2 -526.642} C_VEL
LIN {X 0,Y 608.423,Z 243.689,A -85,B 0,C 180,E1 -529.332,E2 -529.332} C_VEL
LIN {X 0,Y 608.542,Z 257.258,A -85,B 0,C 180,E1 -529.646,E2 -529.646} C_VEL
LIN {X 0,Y 608.53,Z 269.648,A -85,B 0,C 180,E1 -530.066,E2 -530.066} C_VEL
LIN {X 0,Y 608.477,Z 281.512,A -85,B 0,C 180,E1 -530.61,E2 -530.61} C_VEL
LIN {X 0,Y 608.489,Z 292.876,A -85,B 0,C 180,E1 -531.281,E2 -531.281} C_VEL
LIN {X 0,Y 608.494,Z 303.13,A -85,B 0,C 180,E1 -532.033,E2 -532.033} C_VEL
LIN {X 0,Y 608.467,Z 312.365,A -85,B 0,C 180,E1 -532.867,E2 -532.867} C_VEL
LIN {X 0,Y 608.446,Z 321.319,A -85,B 0,C 180,E1 -533.867,E2 -533.867} C_VEL
LIN {X 0,Y 608.446,Z 328.539,A -85,B 0,C 180,E1 -534.864,E2 -534.864} C_VEL
LIN {X 0,Y 608.439,Z 333.414,A -85,B 0,C 180,E1 -535.694,E2 -535.694} C_VEL
LIN {X 0,Y 608.43,Z 338.157,A -85,B 0,C 180,E1 -536.689,E2 -536.689} C_VEL
LIN {X 0,Y 608.43,Z 341.793,A -85,B 0,C 180,E1 -537.683,E2 -537.683} C_VEL
LIN {X 0,Y 608.448,Z 344.428,A -85,B 0,C 180,E1 -538.676,E2 -538.676} C_VEL
LIN {X 0,Y 608.437,Z 346.507,A -85,B 0,C 180,E1 -540,E2 -540} C_VEL
LIN {X 0,Y 608.449,Z 346.941,A -85,B 0,C 180,E1 -541.324,E2 -541.324} C_VEL
LIN {X 0,Y 608.445,Z 346.587,A -85,B 0,C 180,E1 -541.986,E2 -541.986} C_VEL
LIN {X 0,Y 608.422,Z 345.836,A -85,B 0,C 180,E1 -542.648,E2 -542.648} C_VEL
LIN {X 0,Y 608.424,Z 344.65,A -85,B 0,C 180,E1 -543.311,E2 -543.311} C_VEL
LIN {X 0,Y 608.432,Z 342.115,A -85,B 0,C 180,E1 -544.306,E2 -544.306} C_VEL
LIN {X 0,Y 608.441,Z 338.579,A -85,B 0,C 180,E1 -545.302,E2 -545.302} C_VEL
LIN {X 0,Y 608.452,Z 333.566,A -85,B 0,C 180,E1 -546.368,E2 -546.368} C_VEL
LIN {X 0,Y 608.451,Z 326.92,A -85,B 0,C 180,E1 -547.467,E2 -547.467} C_VEL
LIN {X 0,Y 608.464,Z 319.318,A -85,B 0,C 180,E1 -548.469,E2 -548.469} C_VEL
LIN {X 0,Y 608.473,Z 314.714,A -85,B 0,C 180,E1 -548.981,E2 -548.981} C_VEL
LIN {X 0,Y 607.802,Z 310.775,A -85,B 0,C 180,E1 -549.387,E2 -549.387} C_VEL
LIN {X 0,Y 604.942,Z 304.114,A -85,B 0,C 180,E1 -550.029,E2 -550.029} C_VEL
LIN {X 0,Y 602.101,Z 296.997,A -85,B 0,C 180,E1 -550.628,E2 -550.628} C_VEL
LIN {X 0,Y 601.464,Z 292.272,A -85,B 0,C 180,E1 -550.965,E2 -550.965} C_VEL
LIN {X 0,Y 601.498,Z 281.032,A -85,B 0,C 180,E1 -551.628,E2 -551.628} C_VEL
LIN {X 0,Y 601.562,Z 268.876,A -85,B 0,C 180,E1 -552.182,E2 -552.182} C_VEL
LIN {X 0,Y 601.574,Z 256.097,A -85,B 0,C 180,E1 -552.611,E2 -552.611} C_VEL
LIN {X 0,Y 601.392,Z 244.404,A -85,B 0,C 180,E1 -552.883,E2 -552.883} C_VEL
LIN {X 0,Y 601.324,Z 243.663,A -85,B 0,C 180,E1 -552.916,E2 -552.916} C_VEL
LIN {X 0,Y 601.31,Z 239.922,A -85,B 0,C 180,E1 -555.594,E2 -555.594} C_VEL
LIN {X 0,Y 601.308,Z 236.057,A -85,B 0,C 180,E1 -558.396,E2 -558.396} C_VEL
LIN {X 0,Y 601.302,Z 232.188,A -85,B 0,C 180,E1 -561.243,E2 -561.243} C_VEL
LIN {X 0,Y 601.327,Z 228.315,A -85,B 0,C 180,E1 -564.146,E2 -564.146} C_VEL
LIN {X 0,Y 601.32,Z 225.408,A -85,B 0,C 180,E1 -566.368,E2 -566.368} C_VEL
LIN {X 0,Y 601.301,Z 222.456,A -85,B 0,C 180,E1 -568.764,E2 -568.764} C_VEL
LIN {X 0,Y 601.341,Z 219.15,A -85,B 0,C 180,E1 -571.441,E2 -571.441} C_VEL
LIN {X 0,Y 601.367,Z 215.912,A -85,B 0,C 180,E1 -574.123,E2 -574.123} C_VEL
LIN {X 0,Y 601.367,Z 213.931,A -85,B 0,C 180,E1 -575.756,E2 -575.756} C_VEL
LIN {X 0,Y 601.405,Z 213.571,A -85,B 0,C 180,E1 -576.583,E2 -576.583} C_VEL
LIN {X 0,Y 601.419,Z 213.565,A -85,B 0,C 180,E1 -579.126,E2 -579.126} C_VEL
LIN {X 0,Y 601.423,Z 213.573,A -85,B 0,C 180,E1 -581.766,E2 -581.766} C_VEL
LIN {X 0,Y 601.402,Z 213.567,A -85,B 0,C 180,E1 -584.532,E2 -584.532} C_VEL
LIN {X 0,Y 601.387,Z 213.577,A -85,B 0,C 180,E1 -587.412,E2 -587.412} C_VEL
LIN {X 0,Y 601.378,Z 213.57,A -85,B 0,C 180,E1 -590.002,E2 -590.002} C_VEL
LIN {X 0,Y 601.405,Z 213.572,A -85,B 0,C 180,E1 -592.622,E2 -592.622} C_VEL
LIN {X 0,Y 601.406,Z 213.567,A -85,B 0,C 180,E1 -595.88,E2 -595.88} C_VEL
LIN {X 0,Y 601.419,Z 213.572,A -85,B 0,C 180,E1 -598.546,E2 -598.546} C_VEL
LIN {X 0,Y 601.407,Z 213.567,A -85,B 0,C 180,E1 -601.372,E2 -601.372} C_VEL
LIN {X 0,Y 601.411,Z 213.572,A -85,B 0,C 180,E1 -604.134,E2 -604.134} C_VEL
LIN {X 0,Y 601.399,Z 213.568,A -85,B 0,C 180,E1 -606.589,E2 -606.589} C_VEL
LIN {X 0,Y 601.432,Z 213.572,A -85,B 0,C 180,E1 -609.478,E2 -609.478} C_VEL
LIN {X 0,Y 601.394,Z 213.568,A -85,B 0,C 180,E1 -612.311,E2 -612.311} C_VEL
LIN {X 0,Y 601.414,Z 213.567,A -85,B 0,C 180,E1 -614.408,E2 -614.408} C_VEL
LIN {X 0,Y 601.384,Z 213.573,A -85,B 0,C 180,E1 -617.171,E2 -617.171} C_VEL
LIN {X 0,Y 601.423,Z 213.566,A -85,B 0,C 180,E1 -619.905,E2 -619.905} C_VEL
LIN {X 0,Y 601.38,Z 213.575,A -85,B 0,C 180,E1 -622.614,E2 -622.614} C_VEL
LIN {X 0,Y 601.373,Z 213.571,A -85,B 0,C 180,E1 -625.307,E2 -625.307} C_VEL
LIN {X 0,Y 601.435,Z 213.57,A -85,B 0,C 180,E1 -627.991,E2 -627.991} C_VEL
LIN {X 0,Y 601.4,Z 213.567,A -85,B 0,C 180,E1 -630.669,E2 -630.669} C_VEL
LIN {X 0,Y 601.427,Z 213.573,A -85,B 0,C 180,E1 -633.349,E2 -633.349} C_VEL
LIN {X 0,Y 601.402,Z 213.638,A -85,B 0,C 180,E1 -635.112,E2 -635.112} C_VEL
LIN {X 0,Y 601.395,Z 220.811,A -85,B 0,C 180,E1 -638.061,E2 -638.061} C_VEL
LIN {X 0,Y 601.359,Z 227.648,A -85,B 0,C 180,E1 -640.977,E2 -640.977} C_VEL
LIN {X 0,Y 601.381,Z 233.426,A -85,B 0,C 180,E1 -643.517,E2 -643.517} C_VEL
LIN {X 0,Y 601.369,Z 240.595,A -85,B 0,C 180,E1 -646.602,E2 -646.602} C_VEL
LIN {X 0,Y 601.369,Z 246.508,A -85,B 0,C 180,E1 -649.101,E2 -649.101} C_VEL
LIN {X 0,Y 601.34,Z 253.384,A -85,B 0,C 180,E1 -651.962,E2 -651.962} C_VEL
LIN {X 0,Y 601.343,Z 260.492,A -85,B 0,C 180,E1 -654.881,E2 -654.881} C_VEL
LIN {X 0,Y 601.358,Z 267.358,A -85,B 0,C 180,E1 -657.671,E2 -657.671} C_VEL
LIN {X 0,Y 601.501,Z 279.518,A -85,B 0,C 180,E1 -658.005,E2 -658.005} C_VEL
LIN {X 0,Y 601.454,Z 289.303,A -85,B 0,C 180,E1 -658.388,E2 -658.388} C_VEL
LIN {X 0,Y 601.423,Z 297.222,A -85,B 0,C 180,E1 -658.786,E2 -658.786} C_VEL
LIN {X 0,Y 601.431,Z 305.574,A -85,B 0,C 180,E1 -659.308,E2 -659.308} C_VEL
LIN {X 0,Y 601.4,Z 314.041,A -85,B 0,C 180,E1 -659.963,E2 -659.963} C_VEL
LIN {X 0,Y 601.389,Z 322.15,A -85,B 0,C 180,E1 -660.749,E2 -660.749} C_VEL
LIN {X 0,Y 601.377,Z 327.969,A -85,B 0,C 180,E1 -661.447,E2 -661.447} C_VEL
LIN {X 0,Y 601.361,Z 333.821,A -85,B 0,C 180,E1 -662.322,E2 -662.322} C_VEL
LIN {X 0,Y 601.351,Z 338.969,A -85,B 0,C 180,E1 -663.318,E2 -663.318} C_VEL
LIN {X 0,Y 601.342,Z 342.114,A -85,B 0,C 180,E1 -664.124,E2 -664.124} C_VEL
LIN {X 0,Y 601.32,Z 344.84,A -85,B 0,C 180,E1 -665.101,E2 -665.101} C_VEL
LIN {X 0,Y 601.315,Z 346.644,A -85,B 0,C 180,E1 -666.249,E2 -666.249} C_VEL
LIN {X 0,Y 601.332,Z 346.847,A -85,B 0,C 180,E1 -667.427,E2 -667.427} C_VEL
LIN {X 0,Y 601.317,Z 345.836,A -85,B 0,C 180,E1 -668.457,E2 -668.457} C_VEL
LIN {X 0,Y 601.327,Z 343.549,A -85,B 0,C 180,E1 -669.522,E2 -669.522} C_VEL
LIN {X 0,Y 601.335,Z 339.908,A -85,B 0,C 180,E1 -670.564,E2 -670.564} C_VEL
LIN {X 0,Y 601.336,Z 336.837,A -85,B 0,C 180,E1 -671.233,E2 -671.233} C_VEL
LIN {X 0,Y 601.373,Z 331.261,A -85,B 0,C 180,E1 -672.175,E2 -672.175} C_VEL
LIN {X 0,Y 601.399,Z 325.915,A -85,B 0,C 180,E1 -672.9,E2 -672.9} C_VEL
LIN {X 0,Y 601.415,Z 318.592,A -85,B 0,C 180,E1 -673.703,E2 -673.703} C_VEL
LIN {X 0,Y 601.413,Z 310.73,A -85,B 0,C 180,E1 -674.402,E2 -674.402} C_VEL
LIN {X 0,Y 601.456,Z 300.482,A -85,B 0,C 180,E1 -675.118,E2 -675.118} C_VEL
LIN {X 0,Y 601.449,Z 291.524,A -85,B 0,C 180,E1 -675.601,E2 -675.601} C_VEL
LIN {X 0,Y 601.5,Z 283.168,A -85,B 0,C 180,E1 -675.956,E2 -675.956} C_VEL
LIN {X 0,Y 601.492,Z 272.753,A -85,B 0,C 180,E1 -676.282,E2 -676.282} C_VEL
LIN {X 0,Y 601.344,Z 267.317,A -85,B 0,C 180,E1 -676.436,E2 -676.436} C_VEL
LIN {X 0,Y 601.335,Z 259.936,A -85,B 0,C 180,E1 -679.436,E2 -679.436} C_VEL
LIN {X 0,Y 601.325,Z 253.332,A -85,B 0,C 180,E1 -682.15,E2 -682.15} C_VEL
LIN {X 0,Y 601.358,Z 246.331,A -85,B 0,C 180,E1 -685.064,E2 -685.064} C_VEL
LIN {X 0,Y 601.348,Z 240.618,A -85,B 0,C 180,E1 -687.479,E2 -687.479} C_VEL
LIN {X 0,Y 601.341,Z 235.058,A -85,B 0,C 180,E1 -689.866,E2 -689.866} C_VEL
LIN {X 0,Y 601.39,Z 228.16,A -85,B 0,C 180,E1 -692.886,E2 -692.886} C_VEL
LIN {X 0,Y 601.346,Z 222.872,A -85,B 0,C 180,E1 -695.119,E2 -695.119} C_VEL
LIN {X 0,Y 601.377,Z 217.183,A -85,B 0,C 180,E1 -697.404,E2 -697.404} C_VEL
LIN {X 0,Y 601.398,Z 213.575,A -85,B 0,C 180,E1 -698.892,E2 -698.892} C_VEL
LIN {X 0,Y 601.399,Z 213.573,A -85,B 0,C 180,E1 -701.607,E2 -701.607} C_VEL
LIN {X 0,Y 601.415,Z 213.572,A -85,B 0,C 180,E1 -704.409,E2 -704.409} C_VEL
LIN {X 0,Y 601.412,Z 213.574,A -85,B 0,C 180,E1 -707.172,E2 -707.172} C_VEL
LIN {X 0,Y 601.439,Z 213.568,A -85,B 0,C 180,E1 -709.905,E2 -709.905} C_VEL
LIN {X 0,Y 601.445,Z 213.568,A -85,B 0,C 180,E1 -712.615,E2 -712.615} C_VEL
LIN {X 0,Y 601.428,Z 213.573,A -85,B 0,C 180,E1 -715.308,E2 -715.308} C_VEL
LIN {X 0,Y 601.437,Z 213.57,A -85,B 0,C 180,E1 -717.991,E2 -717.991} C_VEL
LIN {X 0,Y 601.438,Z 213.568,A -85,B 0,C 180,E1 -720.669,E2 -720.669} C_VEL
LIN {X 0,Y 601.419,Z 213.571,A -85,B 0,C 180,E1 -723.35,E2 -723.35} C_VEL
LIN {X 0,Y 601.418,Z 213.574,A -85,B 0,C 180,E1 -726.037,E2 -726.037} C_VEL
LIN {X 0,Y 601.413,Z 213.572,A -85,B 0,C 180,E1 -728.738,E2 -728.738} C_VEL
LIN {X 0,Y 601.427,Z 213.569,A -85,B 0,C 180,E1 -731.458,E2 -731.458} C_VEL
LIN {X 0,Y 601.423,Z 213.572,A -85,B 0,C 180,E1 -734.205,E2 -734.205} C_VEL
LIN {X 0,Y 601.425,Z 213.571,A -85,B 0,C 180,E1 -736.986,E2 -736.986} C_VEL
LIN {X 0,Y 601.41,Z 213.572,A -85,B 0,C 180,E1 -739.809,E2 -739.809} C_VEL
LIN {X 0,Y 601.417,Z 213.574,A -85,B 0,C 180,E1 -742.683,E2 -742.683} C_VEL
LIN {X 0,Y 601.402,Z 213.574,A -85,B 0,C 180,E1 -744.879,E2 -744.879} C_VEL
LIN {X 0,Y 601.41,Z 213.574,A -85,B 0,C 180,E1 -747.361,E2 -747.361} C_VEL
LIN {X 0,Y 601.428,Z 213.57,A -85,B 0,C 180,E1 -749.393,E2 -749.393} C_VEL
LIN {X 0,Y 601.405,Z 213.572,A -85,B 0,C 180,E1 -751.727,E2 -751.727} C_VEL
LIN {X 0,Y 601.422,Z 213.57,A -85,B 0,C 180,E1 -754.119,E2 -754.119} C_VEL
LIN {X 0,Y 601.404,Z 213.573,A -85,B 0,C 180,E1 -756.583,E2 -756.583} C_VEL
LIN {X 0,Y 601.416,Z 213.572,A -85,B 0,C 180,E1 -759.126,E2 -759.126} C_VEL
LIN {X 0,Y 601.42,Z 213.574,A -85,B 0,C 180,E1 -761.766,E2 -761.766} C_VEL
LIN {X 0,Y 601.428,Z 213.57,A -85,B 0,C 180,E1 -764.535,E2 -764.535} C_VEL
LIN {X 0,Y 601.419,Z 213.572,A -85,B 0,C 180,E1 -767.409,E2 -767.409} C_VEL
LIN {X 0,Y 601.444,Z 213.568,A -85,B 0,C 180,E1 -770.464,E2 -770.464} C_VEL
LIN {X 0,Y 601.404,Z 213.575,A -85,B 0,C 180,E1 -773.417,E2 -773.417} C_VEL
LIN {X 0,Y 601.453,Z 213.783,A -85,B 0,C 180,E1 -774.16,E2 -774.16} C_VEL
LIN {X 0,Y 601.583,Z 220.824,A -85,B 0,C 180,E1 -776.371,E2 -776.371} C_VEL
LIN {X 0,Y 601.547,Z 229.799,A -85,B 0,C 180,E1 -779.065,E2 -779.065} C_VEL
LIN {X 0,Y 601.451,Z 239.1,A -85,B 0,C 180,E1 -781.755,E2 -781.755} C_VEL
LIN {X 0,Y 601.479,Z 248.394,A -85,B 0,C 180,E1 -784.385,E2 -784.385} C_VEL
LIN {X 0,Y 601.417,Z 257.662,A -85,B 0,C 180,E1 -786.954,E2 -786.954} C_VEL
LIN {X 0,Y 601.427,Z 266.929,A -85,B 0,C 180,E1 -789.478,E2 -789.478} C_VEL
LIN {X 0,Y 601.407,Z 277.52,A -85,B 0,C 180,E1 -792.312,E2 -792.312} C_VEL
LIN {X 0,Y 601.369,Z 288.112,A -85,B 0,C 180,E1 -795.102,E2 -795.102} C_VEL
LIN {X 0,Y 601.348,Z 298.703,A -85,B 0,C 180,E1 -797.856,E2 -797.856} C_VEL
LIN {X 0,Y 601.376,Z 299.53,A -85,B 0,C 180,E1 -798.071,E2 -798.071} C_VEL
LIN {X 0,Y 601.619,Z 311.269,A -85,B 0,C 180,E1 -798.311,E2 -798.311} C_VEL
LIN {X 0,Y 601.533,Z 324.347,A -85,B 0,C 180,E1 -798.691,E2 -798.691} C_VEL
LIN {X 0,Y 601.481,Z 335.242,A -85,B 0,C 180,E1 -799.132,E2 -799.132} C_VEL
LIN {X 0,Y 601.478,Z 346.758,A -85,B 0,C 180,E1 -799.736,E2 -799.736} C_VEL
LIN {X 0,Y 601.462,Z 358.254,A -85,B 0,C 180,E1 -800.5,E2 -800.5} C_VEL
LIN {X 0,Y 601.436,Z 367.537,A -85,B 0,C 180,E1 -801.262,E2 -801.262} C_VEL
LIN {X 0,Y 601.4,Z 375.99,A -85,B 0,C 180,E1 -802.108,E2 -802.108} C_VEL
LIN {X 0,Y 601.382,Z 384.236,A -85,B 0,C 180,E1 -803.12,E2 -803.12} C_VEL
LIN {X 0,Y 601.373,Z 390.877,A -85,B 0,C 180,E1 -804.131,E2 -804.131} C_VEL
LIN {X 0,Y 601.336,Z 396.95,A -85,B 0,C 180,E1 -805.307,E2 -805.307} C_VEL
LIN {X 0,Y 601.368,Z 400.896,A -85,B 0,C 180,E1 -806.315,E2 -806.315} C_VEL
LIN {X 0,Y 601.325,Z 403.809,A -85,B 0,C 180,E1 -807.321,E2 -807.321} C_VEL
LIN {X 0,Y 601.343,Z 405.202,A -85,B 0,C 180,E1 -807.991,E2 -807.991} C_VEL
LIN {X 0,Y 601.339,Z 406.784,A -85,B 0,C 180,E1 -809.33,E2 -809.33} C_VEL
LIN {X 0,Y 601.335,Z 407,A -85,B 0,C 180,E1 -810,E2 -810} C_VEL
LIN {X 0,Y 601.347,Z 406.184,A -85,B 0,C 180,E1 -811.339,E2 -811.339} C_VEL
LIN {X 0,Y 601.343,Z 405.202,A -85,B 0,C 180,E1 -812.009,E2 -812.009} C_VEL
LIN {X 0,Y 601.325,Z 403.809,A -85,B 0,C 180,E1 -812.68,E2 -812.68} C_VEL
LIN {X 0,Y 601.368,Z 400.896,A -85,B 0,C 180,E1 -813.685,E2 -813.685} C_VEL
LIN {X 0,Y 601.336,Z 396.949,A -85,B 0,C 180,E1 -814.693,E2 -814.693} C_VEL
LIN {X 0,Y 601.373,Z 390.876,A -85,B 0,C 180,E1 -815.869,E2 -815.869} C_VEL
LIN {X 0,Y 601.382,Z 384.234,A -85,B 0,C 180,E1 -816.88,E2 -816.88} C_VEL
LIN {X 0,Y 601.4,Z 375.988,A -85,B 0,C 180,E1 -817.892,E2 -817.892} C_VEL
LIN {X 0,Y 601.436,Z 367.535,A -85,B 0,C 180,E1 -818.738,E2 -818.738} C_VEL
LIN {X 0,Y 601.449,Z 357.09,A -85,B 0,C 180,E1 -819.585,E2 -819.585} C_VEL
LIN {X 0,Y 601.478,Z 346.754,A -85,B 0,C 180,E1 -820.264,E2 -820.264} C_VEL
LIN {X 0,Y 601.482,Z 335.232,A -85,B 0,C 180,E1 -820.869,E2 -820.869} C_VEL
LIN {X 0,Y 601.527,Z 322.331,A -85,B 0,C 180,E1 -821.376,E2 -821.376} C_VEL
LIN {X 0,Y 601.617,Z 309.43,A -85,B 0,C 180,E1 -821.732,E2 -821.732} C_VEL
LIN {X 0,Y 601.378,Z 299.529,A -85,B 0,C 180,E1 -821.93,E2 -821.93} C_VEL
LIN {X 0,Y 601.384,Z 289.435,A -85,B 0,C 180,E1 -824.552,E2 -824.552} C_VEL
LIN {X 0,Y 601.395,Z 278.843,A -85,B 0,C 180,E1 -827.338,E2 -827.338} C_VEL
LIN {X 0,Y 601.424,Z 268.252,A -85,B 0,C 180,E1 -830.165,E2 -830.165} C_VEL
LIN {X 0,Y 601.413,Z 258.985,A -85,B 0,C 180,E1 -832.683,E2 -832.683} C_VEL
LIN {X 0,Y 601.454,Z 249.717,A -85,B 0,C 180,E1 -835.246,E2 -835.246} C_VEL
LIN {X 0,Y 601.478,Z 240.45,A -85,B 0,C 180,E1 -837.865,E2 -837.865} C_VEL
LIN {X 0,Y 601.451,Z 232.255,A -85,B 0,C 180,E1 -840.163,E2 -840.163} C_VEL
LIN {X 0,Y 601.545,Z 223.636,A -85,B 0,C 180,E1 -842.733,E2 -842.733} C_VEL
LIN {X 0,Y 601.588,Z 216.958,A -85,B 0,C 180,E1 -844.921,E2 -844.921} C_VEL
LIN {X 0,Y 601.422,Z 213.573,A -85,B 0,C 180,E1 -846.201,E2 -846.201} C_VEL
LIN {X 0,Y 601.415,Z 213.571,A -85,B 0,C 180,E1 -848.469,E2 -848.469} C_VEL
LIN {X 0,Y 601.417,Z 213.571,A -85,B 0,C 180,E1 -850.875,E2 -850.875} C_VEL
LIN {X 0,Y 601.432,Z 213.569,A -85,B 0,C 180,E1 -853.586,E2 -853.586} C_VEL
LIN {X 0,Y 601.433,Z 213.57,A -85,B 0,C 180,E1 -856.427,E2 -856.427} C_VEL
LIN {X 0,Y 601.413,Z 213.574,A -85,B 0,C 180,E1 -859.125,E2 -859.125} C_VEL
LIN {X 0,Y 601.423,Z 213.574,A -85,B 0,C 180,E1 -861.732,E2 -861.732} C_VEL
LIN {X 0,Y 601.391,Z 213.578,A -85,B 0,C 180,E1 -864.245,E2 -864.245} C_VEL
LIN {X 0,Y 601.414,Z 213.571,A -85,B 0,C 180,E1 -865.068,E2 -865.068} C_VEL
LIN {X 0,Y 601.38,Z 214.189,A -85,B 0,C 180,E1 -866.073,E2 -866.073} C_VEL
LIN {X 0,Y 601.37,Z 217.118,A -85,B 0,C 180,E1 -868.554,E2 -868.554} C_VEL
LIN {X 0,Y 601.338,Z 220.352,A -85,B 0,C 180,E1 -871.368,E2 -871.368} C_VEL
LIN {X 0,Y 601.307,Z 222.883,A -85,B 0,C 180,E1 -873.632,E2 -873.632} C_VEL
LIN {X 0,Y 601.307,Z 225.579,A -85,B 0,C 180,E1 -875.853,E2 -875.853} C_VEL
LIN {X 0,Y 601.307,Z 228.439,A -85,B 0,C 180,E1 -878.037,E2 -878.037} C_VEL
LIN {X 0,Y 601.298,Z 231.302,A -85,B 0,C 180,E1 -880.187,E2 -880.187} C_VEL
LIN {X 0,Y 601.319,Z 235.122,A -85,B 0,C 180,E1 -883.011,E2 -883.011} C_VEL
LIN {X 0,Y 601.352,Z 239.145,A -85,B 0,C 180,E1 -885.937,E2 -885.937} C_VEL
LIN {X 0,Y 601.305,Z 242.774,A -85,B 0,C 180,E1 -888.539,E2 -888.539} C_VEL
LIN {X 0,Y 601.342,Z 243.722,A -85,B 0,C 180,E1 -889.194,E2 -889.194} C_VEL
LIN {X 0,Y 601.607,Z 251.254,A -85,B 0,C 180,E1 -889.355,E2 -889.355} C_VEL
LIN {X 0,Y 601.56,Z 264.354,A -85,B 0,C 180,E1 -889.737,E2 -889.737} C_VEL
LIN {X 0,Y 601.513,Z 276.673,A -85,B 0,C 180,E1 -890.246,E2 -890.246} C_VEL
LIN {X 0,Y 601.458,Z 289.141,A -85,B 0,C 180,E1 -890.924,E2 -890.924} C_VEL
LIN {X 0,Y 601.447,Z 300.116,A -85,B 0,C 180,E1 -891.686,E2 -891.686} C_VEL
LIN {X 0,Y 601.412,Z 310.786,A -85,B 0,C 180,E1 -892.615,E2 -892.615} C_VEL
LIN {X 0,Y 601.395,Z 319.858,A -85,B 0,C 180,E1 -893.601,E2 -893.601} C_VEL
LIN {X 0,Y 601.376,Z 327.505,A -85,B 0,C 180,E1 -894.636,E2 -894.636} C_VEL
LIN {X 0,Y 601.356,Z 333.481,A -85,B 0,C 180,E1 -895.643,E2 -895.643} C_VEL
LIN {X 0,Y 601.348,Z 338.209,A -85,B 0,C 180,E1 -896.65,E2 -896.65} C_VEL
LIN {X 0,Y 601.341,Z 341.833,A -85,B 0,C 180,E1 -897.656,E2 -897.656} C_VEL
LIN {X 0,Y 601.348,Z 344.455,A -85,B 0,C 180,E1 -898.661,E2 -898.661} C_VEL
LIN {X 0,Y 601.338,Z 345.686,A -85,B 0,C 180,E1 -899.33,E2 -899.33} C_VEL
LIN {X 0,Y 601.338,Z 346.518,A -85,B 0,C 180,E1 -900,E2 -900} C_VEL
LIN {X 0,Y 601.348,Z 346.938,A -85,B 0,C 180,E1 -901.339,E2 -901.339} C_VEL
LIN {X 0,Y 601.343,Z 346.579,A -85,B 0,C 180,E1 -902.009,E2 -902.009} C_VEL
LIN {X 0,Y 601.321,Z 345.817,A -85,B 0,C 180,E1 -902.68,E2 -902.68} C_VEL
LIN {X 0,Y 601.34,Z 344.624,A -85,B 0,C 180,E1 -903.35,E2 -903.35} C_VEL
LIN {X 0,Y 601.348,Z 342.076,A -85,B 0,C 180,E1 -904.357,E2 -904.357} C_VEL
LIN {X 0,Y 601.356,Z 338.527,A -85,B 0,C 180,E1 -905.365,E2 -905.365} C_VEL
LIN {X 0,Y 601.356,Z 332.719,A -85,B 0,C 180,E1 -906.588,E2 -906.588} C_VEL
LIN {X 0,Y 601.388,Z 325.704,A -85,B 0,C 180,E1 -907.724,E2 -907.724} C_VEL
LIN {X 0,Y 601.407,Z 317.743,A -85,B 0,C 180,E1 -908.738,E2 -908.738} C_VEL
LIN {X 0,Y 601.421,Z 307.839,A -85,B 0,C 180,E1 -909.756,E2 -909.756} C_VEL
LIN {X 0,Y 601.468,Z 297.432,A -85,B 0,C 180,E1 -910.605,E2 -910.605} C_VEL
LIN {X 0,Y 601.464,Z 292.272,A -85,B 0,C 180,E1 -910.965,E2 -910.965} C_VEL
LIN {X 0,Y 600.831,Z 287.427,A -85,B 0,C 180,E1 -911.282,E2 -911.282} C_VEL
LIN {X 0,Y 598.021,Z 279.415,A -85,B 0,C 180,E1 -911.773,E2 -911.773} C_VEL
LIN {X 0,Y 595.279,Z 271.067,A -85,B 0,C 180,E1 -912.211,E2 -912.211} C_VEL
LIN {X 0,Y 594.612,Z 265.696,A -85,B 0,C 180,E1 -912.437,E2 -912.437} C_VEL
LIN {X 0,Y 594.635,Z 253.307,A -85,B 0,C 180,E1 -912.825,E2 -912.825} C_VEL
LIN {X 0,Y 594.507,Z 245.597,A -85,B 0,C 180,E1 -912.999,E2 -912.999} C_VEL
LIN {X 0,Y 594.236,Z 243.675,A -85,B 0,C 180,E1 -913.051,E2 -913.051} C_VEL
LIN {X 0,Y 594.239,Z 239.904,A -85,B 0,C 180,E1 -915.785,E2 -915.785} C_VEL
LIN {X 0,Y 594.237,Z 236.039,A -85,B 0,C 180,E1 -918.622,E2 -918.622} C_VEL
LIN {X 0,Y 594.21,Z 232.169,A -85,B 0,C 180,E1 -921.509,E2 -921.509} C_VEL
LIN {X 0,Y 594.242,Z 228.296,A -85,B 0,C 180,E1 -924.453,E2 -924.453} C_VEL
LIN {X 0,Y 594.24,Z 225.416,A -85,B 0,C 180,E1 -926.707,E2 -926.707} C_VEL
LIN {X 0,Y 594.236,Z 222.694,A -85,B 0,C 180,E1 -929.007,E2 -929.007} C_VEL
LIN {X 0,Y 594.269,Z 219.493,A -85,B 0,C 180,E1 -931.625,E2 -931.625} C_VEL
LIN {X 0,Y 594.298,Z 215.93,A -85,B 0,C 180,E1 -934.586,E2 -934.586} C_VEL
LIN {X 0,Y 594.301,Z 214.94,A -85,B 0,C 180,E1 -935.413,E2 -935.413} C_VEL
LIN {X 0,Y 594.363,Z 214.45,A -85,B 0,C 180,E1 -936.48,E2 -936.48} C_VEL
LIN {X 0,Y 594.385,Z 214.442,A -85,B 0,C 180,E1 -938.805,E2 -938.805} C_VEL
LIN {X 0,Y 594.381,Z 214.451,A -85,B 0,C 180,E1 -941.848,E2 -941.848} C_VEL
LIN {X 0,Y 594.364,Z 214.445,A -85,B 0,C 180,E1 -944.238,E2 -944.238} C_VEL
LIN {X 0,Y 594.344,Z 214.453,A -85,B 0,C 180,E1 -947.151,E2 -947.151} C_VEL
LIN {X 0,Y 594.362,Z 214.449,A -85,B 0,C 180,E1 -949.432,E2 -949.432} C_VEL
LIN {X 0,Y 594.358,Z 214.447,A -85,B 0,C 180,E1 -952.396,E2 -952.396} C_VEL
LIN {X 0,Y 594.358,Z 214.445,A -85,B 0,C 180,E1 -955.418,E2 -955.418} C_VEL
LIN {X 0,Y 594.345,Z 214.448,A -85,B 0,C 180,E1 -957.851,E2 -957.851} C_VEL
LIN {X 0,Y 594.363,Z 214.453,A -85,B 0,C 180,E1 -960.223,E2 -960.223} C_VEL
LIN {X 0,Y 594.38,Z 214.444,A -85,B 0,C 180,E1 -962.539,E2 -962.539} C_VEL
LIN {X 0,Y 594.404,Z 214.445,A -85,B 0,C 180,E1 -965.564,E2 -965.564} C_VEL
LIN {X 0,Y 594.371,Z 214.443,A -85,B 0,C 180,E1 -968.497,E2 -968.497} C_VEL
LIN {X 0,Y 594.379,Z 214.45,A -85,B 0,C 180,E1 -971.382,E2 -971.382} C_VEL
LIN {X 0,Y 594.364,Z 214.444,A -85,B 0,C 180,E1 -974.219,E2 -974.219} C_VEL
LIN {X 0,Y 594.378,Z 214.444,A -85,B 0,C 180,E1 -976.321,E2 -976.321} C_VEL
LIN {X 0,Y 594.351,Z 214.448,A -85,B 0,C 180,E1 -979.094,E2 -979.094} C_VEL
LIN {X 0,Y 594.374,Z 214.445,A -85,B 0,C 180,E1 -981.843,E2 -981.843} C_VEL
LIN {X 0,Y 594.36,Z 214.447,A -85,B 0,C 180,E1 -984.572,E2 -984.572} C_VEL
LIN {X 0,Y 594.372,Z 214.444,A -85,B 0,C 180,E1 -987.289,E2 -987.289} C_VEL
LIN {X 0,Y 594.416,Z 214.442,A -85,B 0,C 180,E1 -990,E2 -990} C_VEL
LIN {X 0,Y 594.387,Z 214.442,A -85,B 0,C 180,E1 -992.711,E2 -992.711} C_VEL
LIN {X 0,Y 594.354,Z 214.46,A -85,B 0,C 180,E1 -995.173,E2 -995.173} C_VEL
LIN {X 0,Y 594.323,Z 220.086,A -85,B 0,C 180,E1 -997.474,E2 -997.474} C_VEL
LIN {X 0,Y 594.311,Z 226.481,A -85,B 0,C 180,E1 -1000.217,E2 -1000.217} C_VEL
LIN {X 0,Y 594.289,Z 232.897,A -85,B 0,C 180,E1 -1002.985,E2 -1002.985} C_VEL
LIN {X 0,Y 594.276,Z 239.293,A -85,B 0,C 180,E1 -1005.783,E2 -1005.783} C_VEL
LIN {X 0,Y 594.279,Z 245.901,A -85,B 0,C 180,E1 -1008.621,E2 -1008.621} C_VEL
LIN {X 0,Y 594.277,Z 252.735,A -85,B 0,C 180,E1 -1011.507,E2 -1011.507} C_VEL
LIN {X 0,Y 594.249,Z 259.811,A -85,B 0,C 180,E1 -1014.452,E2 -1014.452} C_VEL
LIN {X 0,Y 594.275,Z 267.342,A -85,B 0,C 180,E1 -1017.552,E2 -1017.552} C_VEL
LIN {X 0,Y 594.492,Z 279.712,A -85,B 0,C 180,E1 -1017.904,E2 -1017.904} C_VEL
LIN {X 0,Y 594.436,Z 289.042,A -85,B 0,C 180,E1 -1018.272,E2 -1018.272} C_VEL
LIN {X 0,Y 594.401,Z 297.581,A -85,B 0,C 180,E1 -1018.707,E2 -1018.707} C_VEL
LIN {X 0,Y 594.37,Z 306.646,A -85,B 0,C 180,E1 -1019.29,E2 -1019.29} C_VEL
LIN {X 0,Y 594.335,Z 314.91,A -85,B 0,C 180,E1 -1019.954,E2 -1019.954} C_VEL
LIN {X 0,Y 594.313,Z 322.918,A -85,B 0,C 180,E1 -1020.761,E2 -1020.761} C_VEL
LIN {X 0,Y 594.294,Z 329.715,A -85,B 0,C 180,E1 -1021.629,E2 -1021.629} C_VEL
LIN {X 0,Y 594.267,Z 335.279,A -85,B 0,C 180,E1 -1022.523,E2 -1022.523} C_VEL
LIN {X 0,Y 594.258,Z 339.372,A -85,B 0,C 180,E1 -1023.363,E2 -1023.363} C_VEL
LIN {X 0,Y 594.264,Z 342.228,A -85,B 0,C 180,E1 -1024.121,E2 -1024.121} C_VEL
LIN {X 0,Y 594.255,Z 343.671,A -85,B 0,C 180,E1 -1024.588,E2 -1024.588} C_VEL
LIN {X 0,Y 594.222,Z 345.545,A -85,B 0,C 180,E1 -1025.418,E2 -1025.418} C_VEL
LIN {X 0,Y 594.222,Z 346.757,A -85,B 0,C 180,E1 -1026.461,E2 -1026.461} C_VEL
LIN {X 0,Y 594.222,Z 346.994,A -85,B 0,C 180,E1 -1027.099,E2 -1027.099} C_VEL
LIN {X 0,Y 594.219,Z 346.551,A -85,B 0,C 180,E1 -1027.953,E2 -1027.953} C_VEL
LIN {X 0,Y 594.21,Z 345.291,A -85,B 0,C 180,E1 -1028.819,E2 -1028.819} C_VEL
LIN {X 0,Y 594.252,Z 342.934,A -85,B 0,C 180,E1 -1029.759,E2 -1029.759} C_VEL
LIN {X 0,Y 594.241,Z 339.021,A -85,B 0,C 180,E1 -1030.806,E2 -1030.806} C_VEL
LIN {X 0,Y 594.278,Z 333.761,A -85,B 0,C 180,E1 -1031.837,E2 -1031.837} C_VEL
LIN {X 0,Y 594.324,Z 326.921,A -85,B 0,C 180,E1 -1032.847,E2 -1032.847} C_VEL
LIN {X 0,Y 594.35,Z 319.104,A -85,B 0,C 180,E1 -1033.732,E2 -1033.732} C_VEL
LIN {X 0,Y 594.368,Z 310.36,A -85,B 0,C 180,E1 -1034.522,E2 -1034.522} C_VEL
LIN {X 0,Y 594.401,Z 300.013,A -85,B 0,C 180,E1 -1035.242,E2 -1035.242} C_VEL
LIN {X 0,Y 594.434,Z 291.485,A -85,B 0,C 180,E1 -1035.705,E2 -1035.705} C_VEL
LIN {X 0,Y 594.472,Z 281.754,A -85,B 0,C 180,E1 -1036.113,E2 -1036.113} C_VEL
LIN {X 0,Y 594.489,Z 272.526,A -85,B 0,C 180,E1 -1036.398,E2 -1036.398} C_VEL
LIN {X 0,Y 594.271,Z 267.308,A -85,B 0,C 180,E1 -1036.552,E2 -1036.552} C_VEL
LIN {X 0,Y 594.255,Z 260.33,A -85,B 0,C 180,E1 -1039.423,E2 -1039.423} C_VEL
LIN {X 0,Y 594.244,Z 253.151,A -85,B 0,C 180,E1 -1042.41,E2 -1042.41} C_VEL
LIN {X 0,Y 594.293,Z 246.03,A -85,B 0,C 180,E1 -1045.414,E2 -1045.414} C_VEL
LIN {X 0,Y 594.295,Z 239.143,A -85,B 0,C 180,E1 -1048.371,E2 -1048.371} C_VEL
LIN {X 0,Y 594.287,Z 233,A -85,B 0,C 180,E1 -1051.06,E2 -1051.06} C_VEL
LIN {X 0,Y 594.277,Z 227.874,A -85,B 0,C 180,E1 -1053.295,E2 -1053.295} C_VEL
LIN {X 0,Y 594.309,Z 222.292,A -85,B 0,C 180,E1 -1055.584,E2 -1055.584} C_VEL
LIN {X 0,Y 594.296,Z 216.866,A -85,B 0,C 180,E1 -1057.764,E2 -1057.764} C_VEL
LIN {X 0,Y 594.343,Z 214.456,A -85,B 0,C 180,E1 -1058.747,E2 -1058.747} C_VEL
LIN {X 0,Y 594.376,Z 214.449,A -85,B 0,C 180,E1 -1061.382,E2 -1061.382} C_VEL
LIN {X 0,Y 594.368,Z 214.449,A -85,B 0,C 180,E1 -1064.219,E2 -1064.219} C_VEL
LIN {X 0,Y 594.362,Z 214.453,A -85,B 0,C 180,E1 -1067.017,E2 -1067.017} C_VEL
LIN {X 0,Y 594.398,Z 214.446,A -85,B 0,C 180,E1 -1069.784,E2 -1069.784} C_VEL
LIN {X 0,Y 594.398,Z 214.445,A -85,B 0,C 180,E1 -1072.527,E2 -1072.527} C_VEL
LIN {X 0,Y 594.396,Z 214.448,A -85,B 0,C 180,E1 -1075.252,E2 -1075.252} C_VEL
LIN {X 0,Y 594.406,Z 214.446,A -85,B 0,C 180,E1 -1077.967,E2 -1077.967} C_VEL
LIN {X 0,Y 594.411,Z 214.444,A -85,B 0,C 180,E1 -1080.677,E2 -1080.677} C_VEL
LIN {X 0,Y 594.371,Z 214.449,A -85,B 0,C 180,E1 -1083.389,E2 -1083.389} C_VEL
LIN {X 0,Y 594.367,Z 214.452,A -85,B 0,C 180,E1 -1086.109,E2 -1086.109} C_VEL
LIN {X 0,Y 594.379,Z 214.448,A -85,B 0,C 180,E1 -1088.842,E2 -1088.842} C_VEL
LIN {X 0,Y 594.39,Z 214.446,A -85,B 0,C 180,E1 -1091.596,E2 -1091.596} C_VEL
LIN {X 0,Y 594.392,Z 214.449,A -85,B 0,C 180,E1 -1094.377,E2 -1094.377} C_VEL
LIN {X 0,Y 594.387,Z 214.447,A -85,B 0,C 180,E1 -1097.193,E2 -1097.193} C_VEL
LIN {X 0,Y 594.377,Z 214.449,A -85,B 0,C 180,E1 -1100.054,E2 -1100.054} C_VEL
LIN {X 0,Y 594.369,Z 214.45,A -85,B 0,C 180,E1 -1102.967,E2 -1102.967} C_VEL
LIN {X 0,Y 594.376,Z 214.451,A -85,B 0,C 180,E1 -1105.193,E2 -1105.193} C_VEL
LIN {X 0,Y 594.371,Z 214.452,A -85,B 0,C 180,E1 -1107.523,E2 -1107.523} C_VEL
LIN {X 0,Y 594.371,Z 214.449,A -85,B 0,C 180,E1 -1110.325,E2 -1110.325} C_VEL
LIN {X 0,Y 594.38,Z 214.447,A -85,B 0,C 180,E1 -1112.95,E2 -1112.95} C_VEL
LIN {X 0,Y 594.355,Z 214.451,A -85,B 0,C 180,E1 -1115.409,E2 -1115.409} C_VEL
LIN {X 0,Y 594.391,Z 214.447,A -85,B 0,C 180,E1 -1117.94,E2 -1117.94} C_VEL
LIN {X 0,Y 594.379,Z 214.449,A -85,B 0,C 180,E1 -1120.822,E2 -1120.822} C_VEL
LIN {X 0,Y 594.371,Z 214.45,A -85,B 0,C 180,E1 -1123.84,E2 -1123.84} C_VEL
LIN {X 0,Y 594.37,Z 214.45,A -85,B 0,C 180,E1 -1126.701,E2 -1126.701} C_VEL
LIN {X 0,Y 594.367,Z 214.449,A -85,B 0,C 180,E1 -1129.433,E2 -1129.433} C_VEL
LIN {X 0,Y 594.39,Z 214.45,A -85,B 0,C 180,E1 -1132.392,E2 -1132.392} C_VEL
LIN {X 0,Y 594.388,Z 214.574,A -85,B 0,C 180,E1 -1133.915,E2 -1133.915} C_VEL
LIN {X 0,Y 594.616,Z 219.275,A -85,B 0,C 180,E1 -1135.436,E2 -1135.436} C_VEL
LIN {X 0,Y 594.573,Z 227.114,A -85,B 0,C 180,E1 -1137.865,E2 -1137.865} C_VEL
LIN {X 0,Y 594.491,Z 236.315,A -85,B 0,C 180,E1 -1140.619,E2 -1140.619} C_VEL
LIN {X 0,Y 594.443,Z 245.737,A -85,B 0,C 180,E1 -1143.303,E2 -1143.303} C_VEL
LIN {X 0,Y 594.439,Z 255.014,A -85,B 0,C 180,E1 -1145.928,E2 -1145.928} C_VEL
LIN {X 0,Y 594.383,Z 265.498,A -85,B 0,C 180,E1 -1148.832,E2 -1148.832} C_VEL
LIN {X 0,Y 594.379,Z 274.873,A -85,B 0,C 180,E1 -1151.382,E2 -1151.382} C_VEL
LIN {X 0,Y 594.324,Z 285.464,A -85,B 0,C 180,E1 -1154.218,E2 -1154.218} C_VEL
LIN {X 0,Y 594.318,Z 294.731,A -85,B 0,C 180,E1 -1156.668,E2 -1156.668} C_VEL
LIN {X 0,Y 594.288,Z 299.53,A -85,B 0,C 180,E1 -1157.926,E2 -1157.926} C_VEL
LIN {X 0,Y 594.671,Z 305.232,A -85,B 0,C 180,E1 -1158.042,E2 -1158.042} C_VEL
LIN {X 0,Y 594.615,Z 318.498,A -85,B 0,C 180,E1 -1158.365,E2 -1158.365} C_VEL
LIN {X 0,Y 594.53,Z 330.641,A -85,B 0,C 180,E1 -1158.801,E2 -1158.801} C_VEL
LIN {X 0,Y 594.475,Z 342.211,A -85,B 0,C 180,E1 -1159.355,E2 -1159.355} C_VEL
LIN {X 0,Y 594.465,Z 353.478,A -85,B 0,C 180,E1 -1160.043,E2 -1160.043} C_VEL
LIN {X 0,Y 594.406,Z 363.647,A -85,B 0,C 180,E1 -1160.815,E2 -1160.815} C_VEL
LIN {X 0,Y 594.372,Z 372.788,A -85,B 0,C 180,E1 -1161.672,E2 -1161.672} C_VEL
LIN {X 0,Y 594.316,Z 381.691,A -85,B 0,C 180,E1 -1162.697,E2 -1162.697} C_VEL
LIN {X 0,Y 594.281,Z 388.168,A -85,B 0,C 180,E1 -1163.615,E2 -1163.615} C_VEL
LIN {X 0,Y 594.289,Z 393.681,A -85,B 0,C 180,E1 -1164.571,E2 -1164.571} C_VEL
LIN {X 0,Y 594.27,Z 398.372,A -85,B 0,C 180,E1 -1165.591,E2 -1165.591} C_VEL
LIN {X 0,Y 594.267,Z 401.957,A -85,B 0,C 180,E1 -1166.61,E2 -1166.61} C_VEL
LIN {X 0,Y 594.226,Z 403.809,A -85,B 0,C 180,E1 -1167.288,E2 -1167.288} C_VEL
LIN {X 0,Y 594.242,Z 405.201,A -85,B 0,C 180,E1 -1167.967,E2 -1167.967} C_VEL
LIN {X 0,Y 594.239,Z 406.784,A -85,B 0,C 180,E1 -1169.322,E2 -1169.322} C_VEL
LIN {X 0,Y 594.236,Z 407,A -85,B 0,C 180,E1 -1170,E2 -1170} C_VEL
LIN {X 0,Y 594.247,Z 406.185,A -85,B 0,C 180,E1 -1171.355,E2 -1171.355} C_VEL
LIN {X 0,Y 594.242,Z 405.201,A -85,B 0,C 180,E1 -1172.033,E2 -1172.033} C_VEL
LIN {X 0,Y 594.226,Z 403.809,A -85,B 0,C 180,E1 -1172.712,E2 -1172.712} C_VEL
LIN {X 0,Y 594.289,Z 400.896,A -85,B 0,C 180,E1 -1173.729,E2 -1173.729} C_VEL
LIN {X 0,Y 594.241,Z 396.949,A -85,B 0,C 180,E1 -1174.749,E2 -1174.749} C_VEL
LIN {X 0,Y 594.305,Z 390.877,A -85,B 0,C 180,E1 -1175.939,E2 -1175.939} C_VEL
LIN {X 0,Y 594.308,Z 384.235,A -85,B 0,C 180,E1 -1176.962,E2 -1176.962} C_VEL
LIN {X 0,Y 594.359,Z 375.988,A -85,B 0,C 180,E1 -1177.987,E2 -1177.987} C_VEL
LIN {X 0,Y 594.382,Z 367.535,A -85,B 0,C 180,E1 -1178.842,E2 -1178.842} C_VEL
LIN {X 0,Y 594.431,Z 357.091,A -85,B 0,C 180,E1 -1179.7,E2 -1179.7} C_VEL
LIN {X 0,Y 594.454,Z 346.756,A -85,B 0,C 180,E1 -1180.387,E2 -1180.387} C_VEL
LIN {X 0,Y 594.501,Z 334.771,A -85,B 0,C 180,E1 -1181.019,E2 -1181.019} C_VEL
LIN {X 0,Y 594.56,Z 322.486,A -85,B 0,C 180,E1 -1181.505,E2 -1181.505} C_VEL
LIN {X 0,Y 594.676,Z 309.428,A -85,B 0,C 180,E1 -1181.871,E2 -1181.871} C_VEL
LIN {X 0,Y 594.459,Z 300.848,A -85,B 0,C 180,E1 -1182.038,E2 -1182.038} C_VEL
LIN {X 0,Y 594.289,Z 299.529,A -85,B 0,C 180,E1 -1182.074,E2 -1182.074} C_VEL
LIN {X 0,Y 594.313,Z 289.435,A -85,B 0,C 180,E1 -1184.729,E2 -1184.729} C_VEL
LIN {X 0,Y 594.339,Z 278.843,A -85,B 0,C 180,E1 -1187.55,E2 -1187.55} C_VEL
LIN {X 0,Y 594.38,Z 268.252,A -85,B 0,C 180,E1 -1190.415,E2 -1190.415} C_VEL
LIN {X 0,Y 594.406,Z 258.985,A -85,B 0,C 180,E1 -1192.966,E2 -1192.966} C_VEL
LIN {X 0,Y 594.474,Z 249.717,A -85,B 0,C 180,E1 -1195.564,E2 -1195.564} C_VEL
LIN {X 0,Y 594.44,Z 240.216,A -85,B 0,C 180,E1 -1198.224,E2 -1198.224} C_VEL
LIN {X 0,Y 594.466,Z 232.12,A -85,B 0,C 180,E1 -1200.555,E2 -1200.555} C_VEL
LIN {X 0,Y 594.565,Z 224.342,A -85,B 0,C 180,E1 -1202.939,E2 -1202.939} C_VEL
LIN {X 0,Y 594.645,Z 218.33,A -85,B 0,C 180,E1 -1204.962,E2 -1204.962} C_VEL
LIN {X 0,Y 594.376,Z 214.481,A -85,B 0,C 180,E1 -1206.433,E2 -1206.433} C_VEL
LIN {X 0,Y 594.373,Z 214.45,A -85,B 0,C 180,E1 -1208.806,E2 -1208.806} C_VEL
LIN {X 0,Y 594.379,Z 214.45,A -85,B 0,C 180,E1 -1211.848,E2 -1211.848} C_VEL
LIN {X 0,Y 594.36,Z 214.45,A -85,B 0,C 180,E1 -1214.808,E2 -1214.808} C_VEL
LIN {X 0,Y 594.37,Z 214.449,A -85,B 0,C 180,E1 -1217.625,E2 -1217.625} C_VEL
LIN {X 0,Y 594.376,Z 214.45,A -85,B 0,C 180,E1 -1220.319,E2 -1220.319} C_VEL
LIN {X 0,Y 594.387,Z 214.449,A -85,B 0,C 180,E1 -1222.913,E2 -1222.913} C_VEL
LIN {X 0,Y 594.326,Z 214.457,A -85,B 0,C 180,E1 -1225.416,E2 -1225.416} C_VEL
LIN {X 0,Y 594.333,Z 216.174,A -85,B 0,C 180,E1 -1227.096,E2 -1227.096} C_VEL
LIN {X 0,Y 594.29,Z 219.136,A -85,B 0,C 180,E1 -1229.689,E2 -1229.689} C_VEL
LIN {X 0,Y 594.285,Z 222.359,A -85,B 0,C 180,E1 -1232.535,E2 -1232.535} C_VEL
LIN {X 0,Y 594.262,Z 224.849,A -85,B 0,C 180,E1 -1234.802,E2 -1234.802} C_VEL
LIN {X 0,Y 594.229,Z 228.458,A -85,B 0,C 180,E1 -1237.761,E2 -1237.761} C_VEL
LIN {X 0,Y 594.191,Z 232.275,A -85,B 0,C 180,E1 -1240.66,E2 -1240.66} C_VEL
LIN {X 0,Y 594.223,Z 236.096,A -85,B 0,C 180,E1 -1243.51,E2 -1243.51} C_VEL
LIN {X 0,Y 594.245,Z 239.921,A -85,B 0,C 180,E1 -1246.318,E2 -1246.318} C_VEL
LIN {X 0,Y 594.247,Z 243.711,A -85,B 0,C 180,E1 -1249.05,E2 -1249.05} C_VEL
LIN {X 0,Y 594.666,Z 249.006,A -85,B 0,C 180,E1 -1249.164,E2 -1249.164} C_VEL
LIN {X 0,Y 594.624,Z 262.163,A -85,B 0,C 180,E1 -1249.53,E2 -1249.53} C_VEL
LIN {X 0,Y 594.574,Z 273.217,A -85,B 0,C 180,E1 -1249.959,E2 -1249.959} C_VEL
LIN {X 0,Y 594.47,Z 285.095,A -85,B 0,C 180,E1 -1250.559,E2 -1250.559} C_VEL
LIN {X 0,Y 594.436,Z 295.72,A -85,B 0,C 180,E1 -1251.244,E2 -1251.244} C_VEL
LIN {X 0,Y 594.432,Z 305.402,A -85,B 0,C 180,E1 -1252.015,E2 -1252.015} C_VEL
LIN {X 0,Y 594.357,Z 314.227,A -85,B 0,C 180,E1 -1252.868,E2 -1252.868} C_VEL
LIN {X 0,Y 594.329,Z 322.841,A -85,B 0,C 180,E1 -1253.891,E2 -1253.891} C_VEL
LIN {X 0,Y 594.263,Z 329.727,A -85,B 0,C 180,E1 -1254.911,E2 -1254.911} C_VEL
LIN {X 0,Y 594.262,Z 335.245,A -85,B 0,C 180,E1 -1255.931,E2 -1255.931} C_VEL
LIN {X 0,Y 594.277,Z 339.58,A -85,B 0,C 180,E1 -1256.949,E2 -1256.949} C_VEL
LIN {X 0,Y 594.246,Z 342.855,A -85,B 0,C 180,E1 -1257.967,E2 -1257.967} C_VEL
LIN {X 0,Y 594.249,Z 344.482,A -85,B 0,C 180,E1 -1258.645,E2 -1258.645} C_VEL
LIN {X 0,Y 594.239,Z 345.707,A -85,B 0,C 180,E1 -1259.322,E2 -1259.322} C_VEL
LIN {X 0,Y 594.238,Z 346.528,A -85,B 0,C 180,E1 -1260,E2 -1260} C_VEL
LIN {X 0,Y 594.248,Z 346.935,A -85,B 0,C 180,E1 -1261.355,E2 -1261.355} C_VEL
LIN {X 0,Y 594.242,Z 346.569,A -85,B 0,C 180,E1 -1262.033,E2 -1262.033} C_VEL
LIN {X 0,Y 594.222,Z 345.797,A -85,B 0,C 180,E1 -1262.712,E2 -1262.712} C_VEL
LIN {X 0,Y 594.26,Z 344.598,A -85,B 0,C 180,E1 -1263.39,E2 -1263.39} C_VEL
LIN {X 0,Y 594.265,Z 342.038,A -85,B 0,C 180,E1 -1264.409,E2 -1264.409} C_VEL
LIN {X 0,Y 594.277,Z 338.475,A -85,B 0,C 180,E1 -1265.429,E2 -1265.429} C_VEL
LIN {X 0,Y 594.264,Z 333.095,A -85,B 0,C 180,E1 -1266.584,E2 -1266.584} C_VEL
LIN {X 0,Y 594.299,Z 326.754,A -85,B 0,C 180,E1 -1267.645,E2 -1267.645} C_VEL
LIN {X 0,Y 594.356,Z 319.113,A -85,B 0,C 180,E1 -1268.671,E2 -1268.671} C_VEL
LIN {X 0,Y 594.39,Z 309.497,A -85,B 0,C 180,E1 -1269.7,E2 -1269.7} C_VEL
LIN {X 0,Y 594.437,Z 299.567,A -85,B 0,C 180,E1 -1270.56,E2 -1270.56} C_VEL
LIN {X 0,Y 594.461,Z 289.471,A -85,B 0,C 180,E1 -1271.266,E2 -1271.266} C_VEL
LIN {X 0,Y 594.542,Z 277.347,A -85,B 0,C 180,E1 -1271.939,E2 -1271.939} C_VEL
LIN {X 0,Y 594.612,Z 265.696,A -85,B 0,C 180,E1 -1272.437,E2 -1272.437} C_VEL
LIN {X 0,Y 594.112,Z 262.059,A -85,B 0,C 180,E1 -1272.579,E2 -1272.579} C_VEL
LIN {X 0,Y 591.744,Z 256.309,A -85,B 0,C 180,E1 -1272.81,E2 -1272.81} C_VEL
LIN {X 0,Y 588.397,Z 249.334,A -85,B 0,C 180,E1 -1273.051,E2 -1273.051} C_VEL
LIN {X 0,Y 587.625,Z 246.84,A -85,B 0,C 180,E1 -1273.117,E2 -1273.117} C_VEL
LIN {X 0,Y 587.136,Z 243.687,A -85,B 0,C 180,E1 -1273.19,E2 -1273.19} C_VEL
LIN {X 0,Y 587.146,Z 239.886,A -85,B 0,C 180,E1 -1275.98,E2 -1275.98} C_VEL
LIN {X 0,Y 587.138,Z 235.855,A -85,B 0,C 180,E1 -1278.98,E2 -1278.98} C_VEL
LIN {X 0,Y 587.128,Z 232.15,A -85,B 0,C 180,E1 -1281.782,E2 -1281.782} C_VEL
LIN {X 0,Y 587.161,Z 228.277,A -85,B 0,C 180,E1 -1284.767,E2 -1284.767} C_VEL
LIN {X 0,Y 587.186,Z 224.909,A -85,B 0,C 180,E1 -1287.661,E2 -1287.661} C_VEL
LIN {X 0,Y 587.19,Z 221.423,A -85,B 0,C 180,E1 -1290.485,E2 -1290.485} C_VEL
LIN {X 0,Y 587.187,Z 218.31,A -85,B 0,C 180,E1 -1293.088,E2 -1293.088} C_VEL
LIN {X 0,Y 587.218,Z 215.414,A -85,B 0,C 180,E1 -1295.526,E2 -1295.526} C_VEL
LIN {X 0,Y 587.346,Z 215.323,A -85,B 0,C 180,E1 -1297.839,E2 -1297.839} C_VEL
LIN {X 0,Y 587.316,Z 215.327,A -85,B 0,C 180,E1 -1300.255,E2 -1300.255} C_VEL
LIN {X 0,Y 587.309,Z 215.325,A -85,B 0,C 180,E1 -1303.117,E2 -1303.117} C_VEL
LIN {X 0,Y 587.303,Z 215.325,A -85,B 0,C 180,E1 -1306.047,E2 -1306.047} C_VEL
LIN {X 0,Y 587.334,Z 215.325,A -85,B 0,C 180,E1 -1308.926,E2 -1308.926} C_VEL
LIN {X 0,Y 587.296,Z 215.326,A -85,B 0,C 180,E1 -1311.518,E2 -1311.518} C_VEL
LIN {X 0,Y 587.256,Z 215.33,A -85,B 0,C 180,E1 -1314.097,E2 -1314.097} C_VEL
LIN {X 0,Y 587.335,Z 215.323,A -85,B 0,C 180,E1 -1316.89,E2 -1316.89} C_VEL
LIN {X 0,Y 587.322,Z 215.322,A -85,B 0,C 180,E1 -1319.493,E2 -1319.493} C_VEL
LIN {X 0,Y 587.345,Z 215.324,A -85,B 0,C 180,E1 -1322.309,E2 -1322.309} C_VEL
LIN {X 0,Y 587.358,Z 215.321,A -85,B 0,C 180,E1 -1325.42,E2 -1325.42} C_VEL
LIN {X 0,Y 587.328,Z 215.322,A -85,B 0,C 180,E1 -1328.226,E2 -1328.226} C_VEL
LIN {X 0,Y 587.351,Z 215.325,A -85,B 0,C 180,E1 -1331.151,E2 -1331.151} C_VEL
LIN {X 0,Y 587.318,Z 215.322,A -85,B 0,C 180,E1 -1334.024,E2 -1334.024} C_VEL
LIN {X 0,Y 587.355,Z 215.318,A -85,B 0,C 180,E1 -1336.154,E2 -1336.154} C_VEL
LIN {X 0,Y 587.342,Z 215.323,A -85,B 0,C 180,E1 -1338.962,E2 -1338.962} C_VEL
LIN {X 0,Y 587.334,Z 215.321,A -85,B 0,C 180,E1 -1341.744,E2 -1341.744} C_VEL
LIN {X 0,Y 587.329,Z 215.324,A -85,B 0,C 180,E1 -1344.507,E2 -1344.507} C_VEL
LIN {X 0,Y 587.34,Z 215.32,A -85,B 0,C 180,E1 -1347.256,E2 -1347.256} C_VEL
LIN {X 0,Y 587.384,Z 215.318,A -85,B 0,C 180,E1 -1350,E2 -1350} C_VEL
LIN {X 0,Y 587.356,Z 215.318,A -85,B 0,C 180,E1 -1352.743,E2 -1352.743} C_VEL
LIN {X 0,Y 587.297,Z 215.425,A -85,B 0,C 180,E1 -1355.278,E2 -1355.278} C_VEL
LIN {X 0,Y 587.25,Z 222.617,A -85,B 0,C 180,E1 -1358.257,E2 -1358.257} C_VEL
LIN {X 0,Y 587.236,Z 229.068,A -85,B 0,C 180,E1 -1361.075,E2 -1361.075} C_VEL
LIN {X 0,Y 587.251,Z 236.342,A -85,B 0,C 180,E1 -1364.214,E2 -1364.214} C_VEL
LIN {X 0,Y 587.216,Z 242.16,A -85,B 0,C 180,E1 -1366.769,E2 -1366.769} C_VEL
LIN {X 0,Y 587.194,Z 248.669,A -85,B 0,C 180,E1 -1369.58,E2 -1369.58} C_VEL
LIN {X 0,Y 587.172,Z 253.835,A -85,B 0,C 180,E1 -1371.78,E2 -1371.78} C_VEL
LIN {X 0,Y 587.165,Z 260.932,A -85,B 0,C 180,E1 -1374.767,E2 -1374.767} C_VEL
LIN {X 0,Y 587.171,Z 267.38,A -85,B 0,C 180,E1 -1377.449,E2 -1377.449} C_VEL
LIN {X 0,Y 587.499,Z 274.321,A -85,B 0,C 180,E1 -1377.627,E2 -1377.627} C_VEL
LIN {X 0,Y 587.457,Z 285.471,A -85,B 0,C 180,E1 -1378.006,E2 -1378.006} C_VEL
LIN {X 0,Y 587.364,Z 295.715,A -85,B 0,C 180,E1 -1378.497,E2 -1378.497} C_VEL
LIN {X 0,Y 587.325,Z 305.699,A -85,B 0,C 180,E1 -1379.128,E2 -1379.128} C_VEL
LIN {X 0,Y 587.306,Z 313.87,A -85,B 0,C 180,E1 -1379.776,E2 -1379.776} C_VEL
LIN {X 0,Y 587.244,Z 321.2,A -85,B 0,C 180,E1 -1380.494,E2 -1380.494} C_VEL
LIN {X 0,Y 587.24,Z 328.396,A -85,B 0,C 180,E1 -1381.373,E2 -1381.373} C_VEL
LIN {X 0,Y 587.199,Z 333.688,A -85,B 0,C 180,E1 -1382.181,E2 -1382.181} C_VEL
LIN {X 0,Y 587.162,Z 338.35,A -85,B 0,C 180,E1 -1383.085,E2 -1383.085} C_VEL
LIN {X 0,Y 587.161,Z 342.726,A -85,B 0,C 180,E1 -1384.233,E2 -1384.233} C_VEL
LIN {X 0,Y 587.126,Z 344.885,A -85,B 0,C 180,E1 -1385.07,E2 -1385.07} C_VEL
LIN {X 0,Y 587.125,Z 346.269,A -85,B 0,C 180,E1 -1385.912,E2 -1385.912} C_VEL
LIN {X 0,Y 587.126,Z 346.897,A -85,B 0,C 180,E1 -1386.763,E2 -1386.763} C_VEL
LIN {X 0,Y 587.121,Z 346.668,A -85,B 0,C 180,E1 -1387.81,E2 -1387.81} C_VEL
LIN {X 0,Y 587.139,Z 345.124,A -85,B 0,C 180,E1 -1388.918,E2 -1388.918} C_VEL
LIN {X 0,Y 587.161,Z 342.25,A -85,B 0,C 180,E1 -1389.999,E2 -1389.999} C_VEL
LIN {X 0,Y 587.183,Z 338.121,A -85,B 0,C 180,E1 -1391.057,E2 -1391.057} C_VEL
LIN {X 0,Y 587.194,Z 332.591,A -85,B 0,C 180,E1 -1392.092,E2 -1392.092} C_VEL
LIN {X 0,Y 587.233,Z 325.376,A -85,B 0,C 180,E1 -1393.109,E2 -1393.109} C_VEL
LIN {X 0,Y 587.268,Z 317.712,A -85,B 0,C 180,E1 -1393.956,E2 -1393.956} C_VEL
LIN {X 0,Y 587.312,Z 309.303,A -85,B 0,C 180,E1 -1394.696,E2 -1394.696} C_VEL
LIN {X 0,Y 587.362,Z 299.542,A -85,B 0,C 180,E1 -1395.369,E2 -1395.369} C_VEL
LIN {X 0,Y 587.413,Z 290.025,A -85,B 0,C 180,E1 -1395.878,E2 -1395.878} C_VEL
LIN {X 0,Y 587.469,Z 281.432,A -85,B 0,C 180,E1 -1396.234,E2 -1396.234} C_VEL
LIN {X 0,Y 587.493,Z 270.931,A -85,B 0,C 180,E1 -1396.552,E2 -1396.552} C_VEL
LIN {X 0,Y 587.174,Z 267.359,A -85,B 0,C 180,E1 -1396.647,E2 -1396.647} C_VEL
LIN {X 0,Y 587.174,Z 259.951,A -85,B 0,C 180,E1 -1399.734,E2 -1399.734} C_VEL
LIN {X 0,Y 587.16,Z 253.674,A -85,B 0,C 180,E1 -1402.378,E2 -1402.378} C_VEL
LIN {X 0,Y 587.182,Z 247.68,A -85,B 0,C 180,E1 -1404.934,E2 -1404.934} C_VEL
LIN {X 0,Y 587.182,Z 241.955,A -85,B 0,C 180,E1 -1407.411,E2 -1407.411} C_VEL
LIN {X 0,Y 587.229,Z 236.462,A -85,B 0,C 180,E1 -1409.824,E2 -1409.824} C_VEL
LIN {X 0,Y 587.22,Z 229.308,A -85,B 0,C 180,E1 -1412.948,E2 -1412.948} C_VEL
LIN {X 0,Y 587.209,Z 223.229,A -85,B 0,C 180,E1 -1415.451,E2 -1415.451} C_VEL
LIN {X 0,Y 587.229,Z 216.295,A -85,B 0,C 180,E1 -1418.222,E2 -1418.222} C_VEL
LIN {X 0,Y 587.274,Z 215.337,A -85,B 0,C 180,E1 -1418.684,E2 -1418.684} C_VEL
LIN {X 0,Y 587.348,Z 215.327,A -85,B 0,C 180,E1 -1421.151,E2 -1421.151} C_VEL
LIN {X 0,Y 587.324,Z 215.326,A -85,B 0,C 180,E1 -1424.025,E2 -1424.025} C_VEL
LIN {X 0,Y 587.315,Z 215.329,A -85,B 0,C 180,E1 -1426.858,E2 -1426.858} C_VEL
LIN {X 0,Y 587.346,Z 215.325,A -85,B 0,C 180,E1 -1429.66,E2 -1429.66} C_VEL
LIN {X 0,Y 587.371,Z 215.321,A -85,B 0,C 180,E1 -1432.437,E2 -1432.437} C_VEL
LIN {X 0,Y 587.365,Z 215.323,A -85,B 0,C 180,E1 -1435.195,E2 -1435.195} C_VEL
LIN {X 0,Y 587.375,Z 215.322,A -85,B 0,C 180,E1 -1437.943,E2 -1437.943} C_VEL
LIN {X 0,Y 587.383,Z 215.319,A -85,B 0,C 180,E1 -1440.685,E2 -1440.685} C_VEL
LIN {X 0,Y 587.324,Z 215.328,A -85,B 0,C 180,E1 -1443.43,E2 -1443.43} C_VEL
LIN {X 0,Y 587.356,Z 215.322,A -85,B 0,C 180,E1 -1445.493,E2 -1445.493} C_VEL
LIN {X 0,Y 587.368,Z 215.323,A -85,B 0,C 180,E1 -1448.255,E2 -1448.255} C_VEL
LIN {X 0,Y 587.352,Z 215.323,A -85,B 0,C 180,E1 -1451.134,E2 -1451.134} C_VEL
LIN {X 0,Y 587.369,Z 215.323,A -85,B 0,C 180,E1 -1454.26,E2 -1454.26} C_VEL
LIN {X 0,Y 587.35,Z 215.323,A -85,B 0,C 180,E1 -1457.406,E2 -1457.406} C_VEL
LIN {X 0,Y 587.33,Z 215.329,A -85,B 0,C 180,E1 -1460.305,E2 -1460.305} C_VEL
LIN {X 0,Y 587.323,Z 215.326,A -85,B 0,C 180,E1 -1463.259,E2 -1463.259} C_VEL
LIN {X 0,Y 587.342,Z 215.327,A -85,B 0,C 180,E1 -1466.177,E2 -1466.177} C_VEL
LIN {X 0,Y 587.353,Z 215.323,A -85,B 0,C 180,E1 -1469.133,E2 -1469.133} C_VEL
LIN {X 0,Y 587.347,Z 215.324,A -85,B 0,C 180,E1 -1471.836,E2 -1471.836} C_VEL
LIN {X 0,Y 587.346,Z 215.325,A -85,B 0,C 180,E1 -1474.347,E2 -1474.347} C_VEL
LIN {X 0,Y 587.349,Z 215.323,A -85,B 0,C 180,E1 -1477.607,E2 -1477.607} C_VEL
LIN {X 0,Y 587.313,Z 215.328,A -85,B 0,C 180,E1 -1480.255,E2 -1480.255} C_VEL
LIN {X 0,Y 587.316,Z 215.329,A -85,B 0,C 180,E1 -1483.118,E2 -1483.118} C_VEL
LIN {X 0,Y 587.314,Z 215.328,A -85,B 0,C 180,E1 -1486.048,E2 -1486.048} C_VEL
LIN {X 0,Y 587.336,Z 215.328,A -85,B 0,C 180,E1 -1488.925,E2 -1488.925} C_VEL
LIN {X 0,Y 587.327,Z 215.328,A -85,B 0,C 180,E1 -1491.52,E2 -1491.52} C_VEL
LIN {X 0,Y 587.346,Z 215.397,A -85,B 0,C 180,E1 -1493.679,E2 -1493.679} C_VEL
LIN {X 0,Y 587.664,Z 219.29,A -85,B 0,C 180,E1 -1494.967,E2 -1494.967} C_VEL
LIN {X 0,Y 587.617,Z 227.094,A -85,B 0,C 180,E1 -1497.438,E2 -1497.438} C_VEL
LIN {X 0,Y 587.531,Z 234.968,A -85,B 0,C 180,E1 -1499.841,E2 -1499.841} C_VEL
LIN {X 0,Y 587.469,Z 244.441,A -85,B 0,C 180,E1 -1502.623,E2 -1502.623} C_VEL
LIN {X 0,Y 587.432,Z 253.69,A -85,B 0,C 180,E1 -1505.245,E2 -1505.245} C_VEL
LIN {X 0,Y 587.398,Z 262.957,A -85,B 0,C 180,E1 -1507.859,E2 -1507.859} C_VEL
LIN {X 0,Y 587.325,Z 272.225,A -85,B 0,C 180,E1 -1510.424,E2 -1510.424} C_VEL
LIN {X 0,Y 587.283,Z 282.816,A -85,B 0,C 180,E1 -1513.309,E2 -1513.309} C_VEL
LIN {X 0,Y 587.236,Z 293.407,A -85,B 0,C 180,E1 -1516.151,E2 -1516.151} C_VEL
LIN {X 0,Y 587.2,Z 299.572,A -85,B 0,C 180,E1 -1517.789,E2 -1517.789} C_VEL
LIN {X 0,Y 587.741,Z 304.09,A -85,B 0,C 180,E1 -1517.877,E2 -1517.877} C_VEL
LIN {X 0,Y 587.672,Z 317.739,A -85,B 0,C 180,E1 -1518.204,E2 -1518.204} C_VEL
LIN {X 0,Y 587.564,Z 330.421,A -85,B 0,C 180,E1 -1518.657,E2 -1518.657} C_VEL
LIN {X 0,Y 587.477,Z 342.212,A -85,B 0,C 180,E1 -1519.227,E2 -1519.227} C_VEL
LIN {X 0,Y 587.462,Z 353.48,A -85,B 0,C 180,E1 -1519.924,E2 -1519.924} C_VEL
LIN {X 0,Y 587.384,Z 363.647,A -85,B 0,C 180,E1 -1520.705,E2 -1520.705} C_VEL
LIN {X 0,Y 587.34,Z 372.788,A -85,B 0,C 180,E1 -1521.571,E2 -1521.571} C_VEL
LIN {X 0,Y 587.259,Z 381.691,A -85,B 0,C 180,E1 -1522.608,E2 -1522.608} C_VEL
LIN {X 0,Y 587.195,Z 388.745,A -85,B 0,C 180,E1 -1523.627,E2 -1523.627} C_VEL
LIN {X 0,Y 587.211,Z 393.681,A -85,B 0,C 180,E1 -1524.506,E2 -1524.506} C_VEL
LIN {X 0,Y 587.188,Z 398.372,A -85,B 0,C 180,E1 -1525.538,E2 -1525.538} C_VEL
LIN {X 0,Y 587.193,Z 401.957,A -85,B 0,C 180,E1 -1526.569,E2 -1526.569} C_VEL
LIN {X 0,Y 587.132,Z 403.809,A -85,B 0,C 180,E1 -1527.256,E2 -1527.256} C_VEL
LIN {X 0,Y 587.141,Z 405.2,A -85,B 0,C 180,E1 -1527.942,E2 -1527.942} C_VEL
LIN {X 0,Y 587.14,Z 406.784,A -85,B 0,C 180,E1 -1529.314,E2 -1529.314} C_VEL
LIN {X 0,Y 587.137,Z 407,A -85,B 0,C 180,E1 -1530,E2 -1530} C_VEL
LIN {X 0,Y 587.147,Z 406.185,A -85,B 0,C 180,E1 -1531.372,E2 -1531.372} C_VEL
LIN {X 0,Y 587.141,Z 405.201,A -85,B 0,C 180,E1 -1532.058,E2 -1532.058} C_VEL
LIN {X 0,Y 587.132,Z 403.809,A -85,B 0,C 180,E1 -1532.745,E2 -1532.745} C_VEL
LIN {X 0,Y 587.213,Z 400.896,A -85,B 0,C 180,E1 -1533.774,E2 -1533.774} C_VEL
LIN {X 0,Y 587.147,Z 396.949,A -85,B 0,C 180,E1 -1534.806,E2 -1534.806} C_VEL
LIN {X 0,Y 587.218,Z 390.876,A -85,B 0,C 180,E1 -1536.011,E2 -1536.011} C_VEL
LIN {X 0,Y 587.245,Z 384.236,A -85,B 0,C 180,E1 -1537.046,E2 -1537.046} C_VEL
LIN {X 0,Y 587.299,Z 375.989,A -85,B 0,C 180,E1 -1538.083,E2 -1538.083} C_VEL
LIN {X 0,Y 587.343,Z 367.536,A -85,B 0,C 180,E1 -1538.949,E2 -1538.949} C_VEL
LIN {X 0,Y 587.416,Z 357.093,A -85,B 0,C 180,E1 -1539.817,E2 -1539.817} C_VEL
LIN {X 0,Y 587.472,Z 346.755,A -85,B 0,C 180,E1 -1540.512,E2 -1540.512} C_VEL
LIN {X 0,Y 587.53,Z 335.16,A -85,B 0,C 180,E1 -1541.133,E2 -1541.133} C_VEL
LIN {X 0,Y 587.594,Z 322.689,A -85,B 0,C 180,E1 -1541.637,E2 -1541.637} C_VEL
LIN {X 0,Y 587.714,Z 309.427,A -85,B 0,C 180,E1 -1542.014,E2 -1542.014} C_VEL
LIN {X 0,Y 587.494,Z 301.599,A -85,B 0,C 180,E1 -1542.172,E2 -1542.172} C_VEL
LIN {X 0,Y 587.2,Z 299.529,A -85,B 0,C 180,E1 -1542.222,E2 -1542.222} C_VEL
LIN {X 0,Y 587.259,Z 289.435,A -85,B 0,C 180,E1 -1544.91,E2 -1544.91} C_VEL
LIN {X 0,Y 587.304,Z 278.843,A -85,B 0,C 180,E1 -1547.767,E2 -1547.767} C_VEL
LIN {X 0,Y 587.373,Z 268.252,A -85,B 0,C 180,E1 -1550.669,E2 -1550.669} C_VEL
LIN {X 0,Y 587.434,Z 257.661,A -85,B 0,C 180,E1 -1553.628,E2 -1553.628} C_VEL
LIN {X 0,Y 587.438,Z 248.238,A -85,B 0,C 180,E1 -1556.274,E2 -1556.274} C_VEL
LIN {X 0,Y 587.461,Z 238.006,A -85,B 0,C 180,E1 -1559.152,E2 -1559.152} C_VEL
LIN {X 0,Y 587.58,Z 228.045,A -85,B 0,C 180,E1 -1562.177,E2 -1562.177} C_VEL
LIN {X 0,Y 587.687,Z 221.404,A -85,B 0,C 180,E1 -1564.396,E2 -1564.396} C_VEL
LIN {X 0,Y 587.677,Z 217.413,A -85,B 0,C 180,E1 -1565.873,E2 -1565.873} C_VEL
LIN {X 0,Y 587.352,Z 215.326,A -85,B 0,C 180,E1 -1566.747,E2 -1566.747} C_VEL
LIN {X 0,Y 587.33,Z 215.328,A -85,B 0,C 180,E1 -1569.361,E2 -1569.361} C_VEL
LIN {X 0,Y 587.339,Z 215.325,A -85,B 0,C 180,E1 -1572.108,E2 -1572.108} C_VEL
LIN {X 0,Y 587.304,Z 215.329,A -85,B 0,C 180,E1 -1575.087,E2 -1575.087} C_VEL
LIN {X 0,Y 587.328,Z 215.329,A -85,B 0,C 180,E1 -1577.925,E2 -1577.925} C_VEL
LIN {X 0,Y 587.336,Z 215.328,A -85,B 0,C 180,E1 -1580.64,E2 -1580.64} C_VEL
LIN {X 0,Y 587.352,Z 215.325,A -85,B 0,C 180,E1 -1583.293,E2 -1583.293} C_VEL
LIN {X 0,Y 587.274,Z 215.457,A -85,B 0,C 180,E1 -1585.774,E2 -1585.774} C_VEL
LIN {X 0,Y 587.26,Z 218.243,A -85,B 0,C 180,E1 -1588.226,E2 -1588.226} C_VEL
LIN {X 0,Y 587.24,Z 221.208,A -85,B 0,C 180,E1 -1590.887,E2 -1590.887} C_VEL
LIN {X 0,Y 587.195,Z 224.406,A -85,B 0,C 180,E1 -1593.714,E2 -1593.714} C_VEL
LIN {X 0,Y 587.148,Z 226.833,A -85,B 0,C 180,E1 -1595.985,E2 -1595.985} C_VEL
LIN {X 0,Y 587.12,Z 229.431,A -85,B 0,C 180,E1 -1598.218,E2 -1598.218} C_VEL
LIN {X 0,Y 587.136,Z 233.249,A -85,B 0,C 180,E1 -1601.144,E2 -1601.144} C_VEL
LIN {X 0,Y 587.144,Z 237.07,A -85,B 0,C 180,E1 -1604.02,E2 -1604.02} C_VEL
LIN {X 0,Y 587.128,Z 240.896,A -85,B 0,C 180,E1 -1606.854,E2 -1606.854} C_VEL
LIN {X 0,Y 587.139,Z 243.688,A -85,B 0,C 180,E1 -1608.9,E2 -1608.9} C_VEL
LIN {X 0,Y 587.719,Z 248.899,A -85,B 0,C 180,E1 -1609.018,E2 -1609.018} C_VEL
LIN {X 0,Y 587.656,Z 261.787,A -85,B 0,C 180,E1 -1609.379,E2 -1609.379} C_VEL
LIN {X 0,Y 587.602,Z 273.508,A -85,B 0,C 180,E1 -1609.839,E2 -1609.839} C_VEL
LIN {X 0,Y 587.481,Z 285.315,A -85,B 0,C 180,E1 -1610.446,E2 -1610.446} C_VEL
LIN {X 0,Y 587.391,Z 297.056,A -85,B 0,C 180,E1 -1611.225,E2 -1611.225} C_VEL
LIN {X 0,Y 587.361,Z 307.479,A -85,B 0,C 180,E1 -1612.091,E2 -1612.091} C_VEL
LIN {X 0,Y 587.3,Z 315.926,A -85,B 0,C 180,E1 -1612.955,E2 -1612.955} C_VEL
LIN {X 0,Y 587.267,Z 324.167,A -85,B 0,C 180,E1 -1613.989,E2 -1613.989} C_VEL
LIN {X 0,Y 587.233,Z 330.809,A -85,B 0,C 180,E1 -1615.022,E2 -1615.022} C_VEL
LIN {X 0,Y 587.213,Z 336.893,A -85,B 0,C 180,E1 -1616.226,E2 -1616.226} C_VEL
LIN {X 0,Y 587.144,Z 340.849,A -85,B 0,C 180,E1 -1617.256,E2 -1617.256} C_VEL
LIN {X 0,Y 587.148,Z 342.888,A -85,B 0,C 180,E1 -1617.942,E2 -1617.942} C_VEL
LIN {X 0,Y 587.149,Z 344.509,A -85,B 0,C 180,E1 -1618.628,E2 -1618.628} C_VEL
LIN {X 0,Y 587.139,Z 345.727,A -85,B 0,C 180,E1 -1619.314,E2 -1619.314} C_VEL
LIN {X 0,Y 587.139,Z 346.538,A -85,B 0,C 180,E1 -1620,E2 -1620} C_VEL
LIN {X 0,Y 587.148,Z 346.932,A -85,B 0,C 180,E1 -1621.372,E2 -1621.372} C_VEL
LIN {X 0,Y 587.14,Z 346.56,A -85,B 0,C 180,E1 -1622.058,E2 -1622.058} C_VEL
LIN {X 0,Y 587.129,Z 345.777,A -85,B 0,C 180,E1 -1622.744,E2 -1622.744} C_VEL
LIN {X 0,Y 587.183,Z 344.571,A -85,B 0,C 180,E1 -1623.431,E2 -1623.431} C_VEL
LIN {X 0,Y 587.183,Z 341.999,A -85,B 0,C 180,E1 -1624.462,E2 -1624.462} C_VEL
LIN {X 0,Y 587.202,Z 338.423,A -85,B 0,C 180,E1 -1625.495,E2 -1625.495} C_VEL
LIN {X 0,Y 587.18,Z 333.416,A -85,B 0,C 180,E1 -1626.59,E2 -1626.59} C_VEL
LIN {X 0,Y 587.234,Z 326.672,A -85,B 0,C 180,E1 -1627.738,E2 -1627.738} C_VEL
LIN {X 0,Y 587.288,Z 319.007,A -85,B 0,C 180,E1 -1628.776,E2 -1628.776} C_VEL
LIN {X 0,Y 587.353,Z 309.365,A -85,B 0,C 180,E1 -1629.818,E2 -1629.818} C_VEL
LIN {X 0,Y 587.431,Z 299.405,A -85,B 0,C 180,E1 -1630.687,E2 -1630.687} C_VEL
LIN {X 0,Y 587.474,Z 288.138,A -85,B 0,C 180,E1 -1631.472,E2 -1631.472} C_VEL
LIN {X 0,Y 587.579,Z 277.09,A -85,B 0,C 180,E1 -1632.082,E2 -1632.082} C_VEL
LIN {X 0,Y 587.658,Z 264.823,A -85,B 0,C 180,E1 -1632.607,E2 -1632.607} C_VEL
LIN {X 0,Y 587.672,Z 251.855,A -85,B 0,C 180,E1 -1633.002,E2 -1633.002} C_VEL
LIN {X 0,Y 587.625,Z 246.84,A -85,B 0,C 180,E1 -1633.117,E2 -1633.117} C_VEL
LIN {X 0,Y 586.873,Z 244.924,A -85,B 0,C 180,E1 -1633.236,E2 -1633.236} C_VEL
LIN {X 0,Y 585.619,Z 243.432,A -85,B 0,C 180,E1 -1633.501,E2 -1633.501} C_VEL
LIN {X 0,Y 582.872,Z 242.334,A -85,B 0,C 180,E1 -1634.277,E2 -1634.277} C_VEL
LIN {X 0,Y 580.842,Z 241.388,A -85,B 0,C 180,E1 -1635.149,E2 -1635.149} C_VEL
LIN {X 0,Y 580.042,Z 240.061,A -85,B 0,C 180,E1 -1636.037,E2 -1636.037} C_VEL
LIN {X 0,Y 580.061,Z 236.001,A -85,B 0,C 180,E1 -1639.095,E2 -1639.095} C_VEL
LIN {X 0,Y 580.043,Z 233.099,A -85,B 0,C 180,E1 -1641.315,E2 -1641.315} C_VEL
LIN {X 0,Y 580.098,Z 229.334,A -85,B 0,C 180,E1 -1644.325,E2 -1644.325} C_VEL
LIN {X 0,Y 580.098,Z 226.705,A -85,B 0,C 180,E1 -1646.632,E2 -1646.632} C_VEL
LIN {X 0,Y 580.072,Z 223.461,A -85,B 0,C 180,E1 -1649.268,E2 -1649.268} C_VEL
LIN {X 0,Y 580.128,Z 220.179,A -85,B 0,C 180,E1 -1652.002,E2 -1652.002} C_VEL
LIN {X 0,Y 580.152,Z 216.992,A -85,B 0,C 180,E1 -1654.706,E2 -1654.706} C_VEL
LIN {X 0,Y 580.179,Z 216.22,A -85,B 0,C 180,E1 -1655.746,E2 -1655.746} C_VEL
LIN {X 0,Y 580.294,Z 216.205,A -85,B 0,C 180,E1 -1658.146,E2 -1658.146} C_VEL
LIN {X 0,Y 580.302,Z 216.196,A -85,B 0,C 180,E1 -1660.843,E2 -1660.843} C_VEL
LIN {X 0,Y 580.275,Z 216.208,A -85,B 0,C 180,E1 -1663.659,E2 -1663.659} C_VEL
LIN {X 0,Y 580.241,Z 216.204,A -85,B 0,C 180,E1 -1666.614,E2 -1666.614} C_VEL
LIN {X 0,Y 580.296,Z 216.205,A -85,B 0,C 180,E1 -1669.156,E2 -1669.156} C_VEL
LIN {X 0,Y 580.245,Z 216.203,A -85,B 0,C 180,E1 -1671.933,E2 -1671.933} C_VEL
LIN {X 0,Y 580.21,Z 216.212,A -85,B 0,C 180,E1 -1674.449,E2 -1674.449} C_VEL
LIN {X 0,Y 580.286,Z 216.2,A -85,B 0,C 180,E1 -1676.974,E2 -1676.974} C_VEL
LIN {X 0,Y 580.284,Z 216.198,A -85,B 0,C 180,E1 -1679.424,E2 -1679.424} C_VEL
LIN {X 0,Y 580.292,Z 216.205,A -85,B 0,C 180,E1 -1682.143,E2 -1682.143} C_VEL
LIN {X 0,Y 580.326,Z 216.195,A -85,B 0,C 180,E1 -1685.27,E2 -1685.27} C_VEL
LIN {X 0,Y 580.278,Z 216.203,A -85,B 0,C 180,E1 -1687.947,E2 -1687.947} C_VEL
LIN {X 0,Y 580.303,Z 216.199,A -85,B 0,C 180,E1 -1690.913,E2 -1690.913} C_VEL
LIN {X 0,Y 580.268,Z 216.201,A -85,B 0,C 180,E1 -1693.825,E2 -1693.825} C_VEL
LIN {X 0,Y 580.312,Z 216.195,A -85,B 0,C 180,E1 -1695.983,E2 -1695.983} C_VEL
LIN {X 0,Y 580.311,Z 216.201,A -85,B 0,C 180,E1 -1698.827,E2 -1698.827} C_VEL
LIN {X 0,Y 580.302,Z 216.196,A -85,B 0,C 180,E1 -1701.643,E2 -1701.643} C_VEL
LIN {X 0,Y 580.298,Z 216.201,A -85,B 0,C 180,E1 -1704.44,E2 -1704.44} C_VEL
LIN {X 0,Y 580.341,Z 216.199,A -85,B 0,C 180,E1 -1707.918,E2 -1707.918} C_VEL
LIN {X 0,Y 580.353,Z 216.193,A -85,B 0,C 180,E1 -1710,E2 -1710} C_VEL
LIN {X 0,Y 580.325,Z 216.194,A -85,B 0,C 180,E1 -1712.777,E2 -1712.777} C_VEL
LIN {X 0,Y 580.237,Z 216.291,A -85,B 0,C 180,E1 -1715.343,E2 -1715.343} C_VEL
LIN {X 0,Y 580.196,Z 223.517,A -85,B 0,C 180,E1 -1718.358,E2 -1718.358} C_VEL
LIN {X 0,Y 580.179,Z 229.892,A -85,B 0,C 180,E1 -1721.176,E2 -1721.176} C_VEL
LIN {X 0,Y 580.189,Z 237.039,A -85,B 0,C 180,E1 -1724.287,E2 -1724.287} C_VEL
LIN {X 0,Y 580.152,Z 243.045,A -85,B 0,C 180,E1 -1726.902,E2 -1726.902} C_VEL
LIN {X 0,Y 580.103,Z 249.752,A -85,B 0,C 180,E1 -1729.83,E2 -1729.83} C_VEL
LIN {X 0,Y 580.069,Z 254.936,A -85,B 0,C 180,E1 -1732.061,E2 -1732.061} C_VEL
LIN {X 0,Y 580.071,Z 262.057,A -85,B 0,C 180,E1 -1735.091,E2 -1735.091} C_VEL
LIN {X 0,Y 580.095,Z 267.334,A -85,B 0,C 180,E1 -1737.314,E2 -1737.314} C_VEL
LIN {X 0,Y 580.489,Z 274.413,A -85,B 0,C 180,E1 -1737.516,E2 -1737.516} C_VEL
LIN {X 0,Y 580.434,Z 285.127,A -85,B 0,C 180,E1 -1737.883,E2 -1737.883} C_VEL
LIN {X 0,Y 580.348,Z 295.503,A -85,B 0,C 180,E1 -1738.38,E2 -1738.38} C_VEL
LIN {X 0,Y 580.303,Z 304.928,A -85,B 0,C 180,E1 -1738.976,E2 -1738.976} C_VEL
LIN {X 0,Y 580.236,Z 313.364,A -85,B 0,C 180,E1 -1739.642,E2 -1739.642} C_VEL
LIN {X 0,Y 580.201,Z 320.879,A -85,B 0,C 180,E1 -1740.379,E2 -1740.379} C_VEL
LIN {X 0,Y 580.146,Z 327.625,A -85,B 0,C 180,E1 -1741.199,E2 -1741.199} C_VEL
LIN {X 0,Y 580.103,Z 334.2,A -85,B 0,C 180,E1 -1742.213,E2 -1742.213} C_VEL
LIN {X 0,Y 580.087,Z 338.365,A -85,B 0,C 180,E1 -1743.038,E2 -1743.038} C_VEL
LIN {X 0,Y 580.086,Z 341.648,A -85,B 0,C 180,E1 -1743.87,E2 -1743.87} C_VEL
LIN {X 0,Y 580.054,Z 344.117,A -85,B 0,C 180,E1 -1744.712,E2 -1744.712} C_VEL
LIN {X 0,Y 580.027,Z 346.039,A -85,B 0,C 180,E1 -1745.726,E2 -1745.726} C_VEL
LIN {X 0,Y 580.034,Z 346.959,A -85,B 0,C 180,E1 -1746.899,E2 -1746.899} C_VEL
LIN {X 0,Y 580.018,Z 346.305,A -85,B 0,C 180,E1 -1748.167,E2 -1748.167} C_VEL
LIN {X 0,Y 580.046,Z 344.637,A -85,B 0,C 180,E1 -1749.154,E2 -1749.154} C_VEL
LIN {X 0,Y 580.062,Z 341.569,A -85,B 0,C 180,E1 -1750.243,E2 -1750.243} C_VEL
LIN {X 0,Y 580.08,Z 337.18,A -85,B 0,C 180,E1 -1751.308,E2 -1751.308} C_VEL
LIN {X 0,Y 580.13,Z 331.349,A -85,B 0,C 180,E1 -1752.354,E2 -1752.354} C_VEL
LIN {X 0,Y 580.161,Z 323.801,A -85,B 0,C 180,E1 -1753.378,E2 -1753.378} C_VEL
LIN {X 0,Y 580.217,Z 316.655,A -85,B 0,C 180,E1 -1754.146,E2 -1754.146} C_VEL
LIN {X 0,Y 580.293,Z 308.254,A -85,B 0,C 180,E1 -1754.868,E2 -1754.868} C_VEL
LIN {X 0,Y 580.339,Z 299.668,A -85,B 0,C 180,E1 -1755.462,E2 -1755.462} C_VEL
LIN {X 0,Y 580.387,Z 291.639,A -85,B 0,C 180,E1 -1755.908,E2 -1755.908} C_VEL
LIN {X 0,Y 580.465,Z 282.761,A -85,B 0,C 180,E1 -1756.296,E2 -1756.296} C_VEL
LIN {X 0,Y 580.481,Z 272.877,A -85,B 0,C 180,E1 -1756.617,E2 -1756.617} C_VEL
LIN {X 0,Y 580.108,Z 267.354,A -85,B 0,C 180,E1 -1756.767,E2 -1756.767} C_VEL
LIN {X 0,Y 580.094,Z 260.277,A -85,B 0,C 180,E1 -1759.753,E2 -1759.753} C_VEL
LIN {X 0,Y 580.098,Z 253.333,A -85,B 0,C 180,E1 -1762.716,E2 -1762.716} C_VEL
LIN {X 0,Y 580.107,Z 246.97,A -85,B 0,C 180,E1 -1765.469,E2 -1765.469} C_VEL
LIN {X 0,Y 580.143,Z 241.219,A -85,B 0,C 180,E1 -1767.995,E2 -1767.995} C_VEL
LIN {X 0,Y 580.158,Z 234.991,A -85,B 0,C 180,E1 -1770.716,E2 -1770.716} C_VEL
LIN {X 0,Y 580.141,Z 228.968,A -85,B 0,C 180,E1 -1773.37,E2 -1773.37} C_VEL
LIN {X 0,Y 580.145,Z 223.278,A -85,B 0,C 180,E1 -1775.677,E2 -1775.677} C_VEL
LIN {X 0,Y 580.182,Z 216.278,A -85,B 0,C 180,E1 -1778.481,E2 -1778.481} C_VEL
LIN {X 0,Y 580.3,Z 216.203,A -85,B 0,C 180,E1 -1780.913,E2 -1780.913} C_VEL
LIN {X 0,Y 580.274,Z 216.205,A -85,B 0,C 180,E1 -1783.825,E2 -1783.825} C_VEL
LIN {X 0,Y 580.273,Z 216.205,A -85,B 0,C 180,E1 -1786.696,E2 -1786.696} C_VEL
LIN {X 0,Y 580.305,Z 216.203,A -85,B 0,C 180,E1 -1789.533,E2 -1789.533} C_VEL
LIN {X 0,Y 580.333,Z 216.197,A -85,B 0,C 180,E1 -1792.345,E2 -1792.345} C_VEL
LIN {X 0,Y 580.336,Z 216.198,A -85,B 0,C 180,E1 -1795.137,E2 -1795.137} C_VEL
LIN {X 0,Y 580.345,Z 216.198,A -85,B 0,C 180,E1 -1797.918,E2 -1797.918} C_VEL
LIN {X 0,Y 580.356,Z 216.194,A -85,B 0,C 180,E1 -1800.694,E2 -1800.694} C_VEL
LIN {X 0,Y 580.341,Z 216.197,A -85,B 0,C 180,E1 -1802.776,E2 -1802.776} C_VEL
LIN {X 0,Y 580.322,Z 216.199,A -85,B 0,C 180,E1 -1805.56,E2 -1805.56} C_VEL
LIN {X 0,Y 580.331,Z 216.2,A -85,B 0,C 180,E1 -1808.356,E2 -1808.356} C_VEL
LIN {X 0,Y 580.304,Z 216.201,A -85,B 0,C 180,E1 -1811.191,E2 -1811.191} C_VEL
LIN {X 0,Y 580.331,Z 216.198,A -85,B 0,C 180,E1 -1814.017,E2 -1814.017} C_VEL
LIN {X 0,Y 580.316,Z 216.201,A -85,B 0,C 180,E1 -1816.914,E2 -1816.914} C_VEL
LIN {X 0,Y 580.291,Z 216.202,A -85,B 0,C 180,E1 -1819.823,E2 -1819.823} C_VEL
LIN {X 0,Y 580.27,Z 216.205,A -85,B 0,C 180,E1 -1822.053,E2 -1822.053} C_VEL
LIN {X 0,Y 580.292,Z 216.206,A -85,B 0,C 180,E1 -1825.08,E2 -1825.08} C_VEL
LIN {X 0,Y 580.294,Z 216.202,A -85,B 0,C 180,E1 -1827.857,E2 -1827.857} C_VEL
LIN {X 0,Y 580.276,Z 216.205,A -85,B 0,C 180,E1 -1830.693,E2 -1830.693} C_VEL
LIN {X 0,Y 580.286,Z 216.205,A -85,B 0,C 180,E1 -1833.313,E2 -1833.313} C_VEL
LIN {X 0,Y 580.25,Z 216.211,A -85,B 0,C 180,E1 -1835.756,E2 -1835.756} C_VEL
LIN {X 0,Y 580.292,Z 216.206,A -85,B 0,C 180,E1 -1838.146,E2 -1838.146} C_VEL
LIN {X 0,Y 580.3,Z 216.202,A -85,B 0,C 180,E1 -1840.843,E2 -1840.843} C_VEL
LIN {X 0,Y 580.281,Z 216.204,A -85,B 0,C 180,E1 -1843.658,E2 -1843.658} C_VEL
LIN {X 0,Y 580.278,Z 216.207,A -85,B 0,C 180,E1 -1846.609,E2 -1846.609} C_VEL
LIN {X 0,Y 580.3,Z 216.202,A -85,B 0,C 180,E1 -1849.157,E2 -1849.157} C_VEL
LIN {X 0,Y 580.29,Z 216.204,A -85,B 0,C 180,E1 -1851.927,E2 -1851.927} C_VEL
LIN {X 0,Y 580.325,Z 216.28,A -85,B 0,C 180,E1 -1853.458,E2 -1853.458} C_VEL
LIN {X 0,Y 580.71,Z 220.578,A -85,B 0,C 180,E1 -1854.91,E2 -1854.91} C_VEL
LIN {X 0,Y 580.662,Z 228.374,A -85,B 0,C 180,E1 -1857.411,E2 -1857.411} C_VEL
LIN {X 0,Y 580.536,Z 237.552,A -85,B 0,C 180,E1 -1860.241,E2 -1860.241} C_VEL
LIN {X 0,Y 580.427,Z 246.858,A -85,B 0,C 180,E1 -1862.995,E2 -1862.995} C_VEL
LIN {X 0,Y 580.385,Z 256.297,A -85,B 0,C 180,E1 -1865.687,E2 -1865.687} C_VEL
LIN {X 0,Y 580.361,Z 265.605,A -85,B 0,C 180,E1 -1868.325,E2 -1868.325} C_VEL
LIN {X 0,Y 580.279,Z 276.196,A -85,B 0,C 180,E1 -1871.279,E2 -1871.279} C_VEL
LIN {X 0,Y 580.216,Z 286.788,A -85,B 0,C 180,E1 -1874.185,E2 -1874.185} C_VEL
LIN {X 0,Y 580.177,Z 296.055,A -85,B 0,C 180,E1 -1876.694,E2 -1876.694} C_VEL
LIN {X 0,Y 580.125,Z 299.53,A -85,B 0,C 180,E1 -1877.627,E2 -1877.627} C_VEL
LIN {X 0,Y 580.803,Z 305.231,A -85,B 0,C 180,E1 -1877.752,E2 -1877.752} C_VEL
LIN {X 0,Y 580.735,Z 318.499,A -85,B 0,C 180,E1 -1878.083,E2 -1878.083} C_VEL
LIN {X 0,Y 580.598,Z 330.632,A -85,B 0,C 180,E1 -1878.528,E2 -1878.528} C_VEL
LIN {X 0,Y 580.487,Z 342.211,A -85,B 0,C 180,E1 -1879.096,E2 -1879.096} C_VEL
LIN {X 0,Y 580.451,Z 353.481,A -85,B 0,C 180,E1 -1879.801,E2 -1879.801} C_VEL
LIN {X 0,Y 580.352,Z 363.648,A -85,B 0,C 180,E1 -1880.591,E2 -1880.591} C_VEL
LIN {X 0,Y 580.279,Z 372.787,A -85,B 0,C 180,E1 -1881.468,E2 -1881.468} C_VEL
LIN {X 0,Y 580.199,Z 381.69,A -85,B 0,C 180,E1 -1882.518,E2 -1882.518} C_VEL
LIN {X 0,Y 580.12,Z 388.465,A -85,B 0,C 180,E1 -1883.505,E2 -1883.505} C_VEL
LIN {X 0,Y 580.139,Z 393.68,A -85,B 0,C 180,E1 -1884.439,E2 -1884.439} C_VEL
LIN {X 0,Y 580.108,Z 398.372,A -85,B 0,C 180,E1 -1885.484,E2 -1885.484} C_VEL
LIN {X 0,Y 580.123,Z 401.957,A -85,B 0,C 180,E1 -1886.527,E2 -1886.527} C_VEL
LIN {X 0,Y 580.043,Z 403.809,A -85,B 0,C 180,E1 -1887.222,E2 -1887.222} C_VEL
LIN {X 0,Y 580.04,Z 405.199,A -85,B 0,C 180,E1 -1887.917,E2 -1887.917} C_VEL
LIN {X 0,Y 580.04,Z 406.785,A -85,B 0,C 180,E1 -1889.306,E2 -1889.306} C_VEL
LIN {X 0,Y 580.037,Z 407,A -85,B 0,C 180,E1 -1890,E2 -1890} C_VEL
LIN {X 0,Y 580.047,Z 406.186,A -85,B 0,C 180,E1 -1891.389,E2 -1891.389} C_VEL
LIN {X 0,Y 580.04,Z 405.2,A -85,B 0,C 180,E1 -1892.083,E2 -1892.083} C_VEL
LIN {X 0,Y 580.043,Z 403.809,A -85,B 0,C 180,E1 -1892.778,E2 -1892.778} C_VEL
LIN {X 0,Y 580.11,Z 400.895,A -85,B 0,C 180,E1 -1893.821,E2 -1893.821} C_VEL
LIN {X 0,Y 580.053,Z 396.949,A -85,B 0,C 180,E1 -1894.865,E2 -1894.865} C_VEL
LIN {X 0,Y 580.139,Z 390.876,A -85,B 0,C 180,E1 -1896.085,E2 -1896.085} C_VEL
LIN {X 0,Y 580.184,Z 384.236,A -85,B 0,C 180,E1 -1897.133,E2 -1897.133} C_VEL
LIN {X 0,Y 580.25,Z 375.989,A -85,B 0,C 180,E1 -1898.182,E2 -1898.182} C_VEL
LIN {X 0,Y 580.308,Z 367.536,A -85,B 0,C 180,E1 -1899.059,E2 -1899.059} C_VEL
LIN {X 0,Y 580.417,Z 357.094,A -85,B 0,C 180,E1 -1899.936,E2 -1899.936} C_VEL
LIN {X 0,Y 580.474,Z 346.753,A -85,B 0,C 180,E1 -1900.64,E2 -1900.64} C_VEL
LIN {X 0,Y 580.564,Z 335.586,A -85,B 0,C 180,E1 -1901.248,E2 -1901.248} C_VEL
LIN {X 0,Y 580.635,Z 323.762,A -85,B 0,C 180,E1 -1901.742,E2 -1901.742} C_VEL
LIN {X 0,Y 580.768,Z 310.341,A -85,B 0,C 180,E1 -1902.138,E2 -1902.138} C_VEL
LIN {X 0,Y 580.564,Z 302.32,A -85,B 0,C 180,E1 -1902.308,E2 -1902.308} C_VEL
LIN {X 0,Y 580.126,Z 299.529,A -85,B 0,C 180,E1 -1902.373,E2 -1902.373} C_VEL
LIN {X 0,Y 580.219,Z 289.435,A -85,B 0,C 180,E1 -1905.095,E2 -1905.095} C_VEL
LIN {X 0,Y 580.255,Z 278.843,A -85,B 0,C 180,E1 -1907.99,E2 -1907.99} C_VEL
LIN {X 0,Y 580.333,Z 268.49,A -85,B 0,C 180,E1 -1910.865,E2 -1910.865} C_VEL
LIN {X 0,Y 580.405,Z 258.985,A -85,B 0,C 180,E1 -1913.553,E2 -1913.553} C_VEL
LIN {X 0,Y 580.405,Z 248.862,A -85,B 0,C 180,E1 -1916.356,E2 -1916.356} C_VEL
LIN {X 0,Y 580.468,Z 238.519,A -85,B 0,C 180,E1 -1919.338,E2 -1919.338} C_VEL
LIN {X 0,Y 580.595,Z 229.335,A -85,B 0,C 180,E1 -1922.182,E2 -1922.182} C_VEL
LIN {X 0,Y 580.722,Z 222.101,A -85,B 0,C 180,E1 -1924.667,E2 -1924.667} C_VEL
LIN {X 0,Y 580.749,Z 219.07,A -85,B 0,C 180,E1 -1925.825,E2 -1925.825} C_VEL
LIN {X 0,Y 580.308,Z 216.203,A -85,B 0,C 180,E1 -1927.12,E2 -1927.12} C_VEL
LIN {X 0,Y 580.292,Z 216.205,A -85,B 0,C 180,E1 -1930.27,E2 -1930.27} C_VEL
LIN {X 0,Y 580.28,Z 216.206,A -85,B 0,C 180,E1 -1932.707,E2 -1932.707} C_VEL
LIN {X 0,Y 580.262,Z 216.209,A -85,B 0,C 180,E1 -1935.611,E2 -1935.611} C_VEL
LIN {X 0,Y 580.284,Z 216.205,A -85,B 0,C 180,E1 -1938.231,E2 -1938.231} C_VEL
LIN {X 0,Y 580.283,Z 216.204,A -85,B 0,C 180,E1 -1940.965,E2 -1940.965} C_VEL
LIN {X 0,Y 580.272,Z 216.205,A -85,B 0,C 180,E1 -1943.596,E2 -1943.596} C_VEL
LIN {X 0,Y 580.256,Z 216.21,A -85,B 0,C 180,E1 -1945.448,E2 -1945.448} C_VEL
LIN {X 0,Y 580.223,Z 218.771,A -85,B 0,C 180,E1 -1947.983,E2 -1947.983} C_VEL
LIN {X 0,Y 580.189,Z 222.104,A -85,B 0,C 180,E1 -1951.018,E2 -1951.018} C_VEL
LIN {X 0,Y 580.127,Z 225.072,A -85,B 0,C 180,E1 -1953.7,E2 -1953.7} C_VEL
LIN {X 0,Y 580.097,Z 227.26,A -85,B 0,C 180,E1 -1955.675,E2 -1955.675} C_VEL
LIN {X 0,Y 580.057,Z 229.626,A -85,B 0,C 180,E1 -1957.939,E2 -1957.939} C_VEL
LIN {X 0,Y 580.03,Z 232.313,A -85,B 0,C 180,E1 -1960.168,E2 -1960.168} C_VEL
LIN {X 0,Y 580.048,Z 236.238,A -85,B 0,C 180,E1 -1963.174,E2 -1963.174} C_VEL
LIN {X 0,Y 580.084,Z 239.957,A -85,B 0,C 180,E1 -1965.977,E2 -1965.977} C_VEL
LIN {X 0,Y 580.058,Z 243.689,A -85,B 0,C 180,E1 -1968.751,E2 -1968.751} C_VEL
LIN {X 0,Y 580.795,Z 250.066,A -85,B 0,C 180,E1 -1968.901,E2 -1968.901} C_VEL
LIN {X 0,Y 580.717,Z 263.318,A -85,B 0,C 180,E1 -1969.29,E2 -1969.29} C_VEL
LIN {X 0,Y 580.628,Z 273.8,A -85,B 0,C 180,E1 -1969.716,E2 -1969.716} C_VEL
LIN {X 0,Y 580.504,Z 285.528,A -85,B 0,C 180,E1 -1970.33,E2 -1970.33} C_VEL
LIN {X 0,Y 580.374,Z 297.229,A -85,B 0,C 180,E1 -1971.118,E2 -1971.118} C_VEL
LIN {X 0,Y 580.339,Z 307.619,A -85,B 0,C 180,E1 -1971.995,E2 -1971.995} C_VEL
LIN {X 0,Y 580.249,Z 316.036,A -85,B 0,C 180,E1 -1972.868,E2 -1972.868} C_VEL
LIN {X 0,Y 580.21,Z 324.259,A -85,B 0,C 180,E1 -1973.916,E2 -1973.916} C_VEL
LIN {X 0,Y 580.096,Z 329.877,A -85,B 0,C 180,E1 -1974.787,E2 -1974.787} C_VEL
LIN {X 0,Y 580.108,Z 335.364,A -85,B 0,C 180,E1 -1975.832,E2 -1975.832} C_VEL
LIN {X 0,Y 580.094,Z 339.672,A -85,B 0,C 180,E1 -1976.875,E2 -1976.875} C_VEL
LIN {X 0,Y 580.05,Z 342.921,A -85,B 0,C 180,E1 -1977.917,E2 -1977.917} C_VEL
LIN {X 0,Y 580.049,Z 344.536,A -85,B 0,C 180,E1 -1978.612,E2 -1978.612} C_VEL
LIN {X 0,Y 580.04,Z 345.748,A -85,B 0,C 180,E1 -1979.306,E2 -1979.306} C_VEL
LIN {X 0,Y 580.04,Z 346.546,A -85,B 0,C 180,E1 -1980,E2 -1980} C_VEL
LIN {X 0,Y 580.047,Z 346.929,A -85,B 0,C 180,E1 -1981.389,E2 -1981.389} C_VEL
LIN {X 0,Y 580.039,Z 346.55,A -85,B 0,C 180,E1 -1982.083,E2 -1982.083} C_VEL
LIN {X 0,Y 580.04,Z 345.757,A -85,B 0,C 180,E1 -1982.778,E2 -1982.778} C_VEL
LIN {X 0,Y 580.109,Z 344.545,A -85,B 0,C 180,E1 -1983.473,E2 -1983.473} C_VEL
LIN {X 0,Y 580.102,Z 341.96,A -85,B 0,C 180,E1 -1984.517,E2 -1984.517} C_VEL
LIN {X 0,Y 580.127,Z 338.37,A -85,B 0,C 180,E1 -1985.562,E2 -1985.562} C_VEL
LIN {X 0,Y 580.126,Z 332.92,A -85,B 0,C 180,E1 -1986.753,E2 -1986.753} C_VEL
LIN {X 0,Y 580.166,Z 326.59,A -85,B 0,C 180,E1 -1987.833,E2 -1987.833} C_VEL
LIN {X 0,Y 580.226,Z 318.9,A -85,B 0,C 180,E1 -1988.884,E2 -1988.884} C_VEL
LIN {X 0,Y 580.294,Z 309.232,A -85,B 0,C 180,E1 -1989.938,E2 -1989.938} C_VEL
LIN {X 0,Y 580.407,Z 299.372,A -85,B 0,C 180,E1 -1990.807,E2 -1990.807} C_VEL
LIN {X 0,Y 580.461,Z 288.35,A -85,B 0,C 180,E1 -1991.586,E2 -1991.586} C_VEL
LIN {X 0,Y 580.59,Z 276.826,A -85,B 0,C 180,E1 -1992.23,E2 -1992.23} C_VEL
LIN {X 0,Y 580.7,Z 264.474,A -85,B 0,C 180,E1 -1992.76,E2 -1992.76} C_VEL
LIN {X 0,Y 580.739,Z 251.315,A -85,B 0,C 180,E1 -1993.16,E2 -1993.16} C_VEL
LIN {X 0,Y 580.469,Z 246.522,A -85,B 0,C 180,E1 -1993.275,E2 -1993.275} C_VEL
LIN {X 0,Y 580.075,Z 243.669,A -85,B 0,C 180,E1 -1993.353,E2 -1993.353} C_VEL
LIN {X 0,Y 580.042,Z 240.061,A -85,B 0,C 180,E1 -1996.037,E2 -1996.037} C_VEL
LIN {X 0,Y 579.385,Z 239.317,A -85,B 0,C 180,E1 -1996.612,E2 -1996.612} C_VEL
LIN {X 0,Y 576.497,Z 238.188,A -85,B 0,C 180,E1 -1997.545,E2 -1997.545} C_VEL
LIN {X 0,Y 574.058,Z 237.298,A -85,B 0,C 180,E1 -1998.297,E2 -1998.297} C_VEL
LIN {X 0,Y 573.028,Z 236.583,A -85,B 0,C 180,E1 -1998.877,E2 -1998.877} C_VEL
LIN {X 0,Y 572.955,Z 236.331,A -85,B 0,C 180,E1 -1999.073,E2 -1999.073} C_VEL
LIN {X 0,Y 572.936,Z 233.083,A -85,B 0,C 180,E1 -2001.592,E2 -2001.592} C_VEL
LIN {X 0,Y 572.98,Z 230.421,A -85,B 0,C 180,E1 -2003.877,E2 -2003.877} C_VEL
LIN {X 0,Y 573.042,Z 227.44,A -85,B 0,C 180,E1 -2006.452,E2 -2006.452} C_VEL
LIN {X 0,Y 573.006,Z 224.84,A -85,B 0,C 180,E1 -2008.577,E2 -2008.577} C_VEL
LIN {X 0,Y 573.04,Z 221.958,A -85,B 0,C 180,E1 -2011.005,E2 -2011.005} C_VEL
LIN {X 0,Y 573.062,Z 218.997,A -85,B 0,C 180,E1 -2013.496,E2 -2013.496} C_VEL
LIN {X 0,Y 573.085,Z 217.104,A -85,B 0,C 180,E1 -2015.197,E2 -2015.197} C_VEL
LIN {X 0,Y 573.238,Z 217.08,A -85,B 0,C 180,E1 -2017.808,E2 -2017.808} C_VEL
LIN {X 0,Y 573.25,Z 217.076,A -85,B 0,C 180,E1 -2020.525,E2 -2020.525} C_VEL
LIN {X 0,Y 573.236,Z 217.081,A -85,B 0,C 180,E1 -2023.36,E2 -2023.36} C_VEL
LIN {X 0,Y 573.211,Z 217.079,A -85,B 0,C 180,E1 -2026.335,E2 -2026.335} C_VEL
LIN {X 0,Y 573.25,Z 217.079,A -85,B 0,C 180,E1 -2029.475,E2 -2029.475} C_VEL
LIN {X 0,Y 573.196,Z 217.081,A -85,B 0,C 180,E1 -2032.189,E2 -2032.189} C_VEL
LIN {X 0,Y 573.217,Z 217.08,A -85,B 0,C 180,E1 -2035.232,E2 -2035.232} C_VEL
LIN {X 0,Y 573.24,Z 217.076,A -85,B 0,C 180,E1 -2037.774,E2 -2037.774} C_VEL
LIN {X 0,Y 573.245,Z 217.078,A -85,B 0,C 180,E1 -2040.633,E2 -2040.633} C_VEL
LIN {X 0,Y 573.213,Z 217.079,A -85,B 0,C 180,E1 -2043.022,E2 -2043.022} C_VEL
LIN {X 0,Y 573.279,Z 217.074,A -85,B 0,C 180,E1 -2045.366,E2 -2045.366} C_VEL
LIN {X 0,Y 573.235,Z 217.077,A -85,B 0,C 180,E1 -2048.419,E2 -2048.419} C_VEL
LIN {X 0,Y 573.274,Z 217.073,A -85,B 0,C 180,E1 -2050.731,E2 -2050.731} C_VEL
LIN {X 0,Y 573.244,Z 217.077,A -85,B 0,C 180,E1 -2053.621,E2 -2053.621} C_VEL
LIN {X 0,Y 573.256,Z 217.074,A -85,B 0,C 180,E1 -2055.806,E2 -2055.806} C_VEL
LIN {X 0,Y 573.268,Z 217.079,A -85,B 0,C 180,E1 -2058.745,E2 -2058.745} C_VEL
LIN {X 0,Y 573.246,Z 217.075,A -85,B 0,C 180,E1 -2061.54,E2 -2061.54} C_VEL
LIN {X 0,Y 573.266,Z 217.078,A -85,B 0,C 180,E1 -2064.371,E2 -2064.371} C_VEL
LIN {X 0,Y 573.31,Z 217.075,A -85,B 0,C 180,E1 -2067.892,E2 -2067.892} C_VEL
LIN {X 0,Y 573.322,Z 217.069,A -85,B 0,C 180,E1 -2070,E2 -2070} C_VEL
LIN {X 0,Y 573.294,Z 217.07,A -85,B 0,C 180,E1 -2072.811,E2 -2072.811} C_VEL
LIN {X 0,Y 573.155,Z 217.108,A -85,B 0,C 180,E1 -2075.387,E2 -2075.387} C_VEL
LIN {X 0,Y 573.138,Z 222.701,A -85,B 0,C 180,E1 -2077.752,E2 -2077.752} C_VEL
LIN {X 0,Y 573.068,Z 229.209,A -85,B 0,C 180,E1 -2080.6,E2 -2080.6} C_VEL
LIN {X 0,Y 573.082,Z 234.135,A -85,B 0,C 180,E1 -2082.753,E2 -2082.753} C_VEL
LIN {X 0,Y 573.065,Z 239.193,A -85,B 0,C 180,E1 -2084.924,E2 -2084.924} C_VEL
LIN {X 0,Y 573.089,Z 244.129,A -85,B 0,C 180,E1 -2087.117,E2 -2087.117} C_VEL
LIN {X 0,Y 573.015,Z 250.837,A -85,B 0,C 180,E1 -2090.085,E2 -2090.085} C_VEL
LIN {X 0,Y 572.974,Z 256.038,A -85,B 0,C 180,E1 -2092.349,E2 -2092.349} C_VEL
LIN {X 0,Y 573.001,Z 261.774,A -85,B 0,C 180,E1 -2094.82,E2 -2094.82} C_VEL
LIN {X 0,Y 573.019,Z 267.389,A -85,B 0,C 180,E1 -2097.21,E2 -2097.21} C_VEL
LIN {X 0,Y 573.498,Z 274.727,A -85,B 0,C 180,E1 -2097.407,E2 -2097.407} C_VEL
LIN {X 0,Y 573.418,Z 286.143,A -85,B 0,C 180,E1 -2097.811,E2 -2097.811} C_VEL
LIN {X 0,Y 573.336,Z 297.637,A -85,B 0,C 180,E1 -2098.4,E2 -2098.4} C_VEL
LIN {X 0,Y 573.264,Z 306.142,A -85,B 0,C 180,E1 -2098.964,E2 -2098.964} C_VEL
LIN {X 0,Y 573.173,Z 314.951,A -85,B 0,C 180,E1 -2099.698,E2 -2099.698} C_VEL
LIN {X 0,Y 573.133,Z 321.654,A -85,B 0,C 180,E1 -2100.386,E2 -2100.386} C_VEL
LIN {X 0,Y 573.072,Z 328.199,A -85,B 0,C 180,E1 -2101.208,E2 -2101.208} C_VEL
LIN {X 0,Y 573.014,Z 334.409,A -85,B 0,C 180,E1 -2102.19,E2 -2102.19} C_VEL
LIN {X 0,Y 572.991,Z 338.731,A -85,B 0,C 180,E1 -2103.072,E2 -2103.072} C_VEL
LIN {X 0,Y 573.009,Z 341.95,A -85,B 0,C 180,E1 -2103.922,E2 -2103.922} C_VEL
LIN {X 0,Y 572.973,Z 344.232,A -85,B 0,C 180,E1 -2104.733,E2 -2104.733} C_VEL
LIN {X 0,Y 572.947,Z 345.293,A -85,B 0,C 180,E1 -2105.206,E2 -2105.206} C_VEL
